LIN {X 0,Y 364.081,Z 519.091,A -85,B 0,C 180,E1 -13381.398,E2 -13381.398} C_VEL
LIN {X 0,Y 365.841,Z 526.741,A -85,B 0,C 180,E1 -13382.545,E2 -13382.545} C_VEL
LIN {X 0,Y 366.269,Z 538.243,A -85,B 0,C 180,E1 -13383.711,E2 -13383.711} C_VEL
LIN {X 0,Y 365.89,Z 556.59,A -85,B 0,C 180,E1 -13385.171,E2 -13385.171} C_VEL
LIN {X 0,Y 365.376,Z 561.748,A -85,B 0,C 180,E1 -13385.4,E2 -13385.4} C_VEL
LIN {X 0,Y 363.138,Z 602.546,A -85,B 0,C 180,E1 -13386.738,E2 -13386.738} C_VEL
LIN {X 0,Y 361.511,Z 662.702,A -85,B 0,C 180,E1 -13388.248,E2 -13388.248} C_VEL
LIN {X 0,Y 360.674,Z 677.145,A -85,B 0,C 180,E1 -13388.833,E2 -13388.833} C_VEL
LIN {X 0,Y 359.879,Z 691.511,A -85,B 0,C 180,E1 -13389.662,E2 -13389.662} C_VEL
LIN {X 0,Y 358.872,Z 705.143,A -85,B 0,C 180,E1 -13390.702,E2 -13390.702} C_VEL
LIN {X 0,Y 357.508,Z 721.974,A -85,B 0,C 180,E1 -13392.26,E2 -13392.26} C_VEL
LIN {X 0,Y 356.635,Z 733.015,A -85,B 0,C 180,E1 -13393.544,E2 -13393.544} C_VEL
LIN {X 0,Y 355.719,Z 743.896,A -85,B 0,C 180,E1 -13395.117,E2 -13395.117} C_VEL
LIN {X 0,Y 355.107,Z 752.022,A -85,B 0,C 180,E1 -13396.553,E2 -13396.553} C_VEL
LIN {X 0,Y 354.444,Z 759.998,A -85,B 0,C 180,E1 -13398.274,E2 -13398.274} C_VEL
LIN {X 0,Y 353.811,Z 767.392,A -85,B 0,C 180,E1 -13400.28,E2 -13400.28} C_VEL
LIN {X 0,Y 353.542,Z 772.311,A -85,B 0,C 180,E1 -13402.001,E2 -13402.001} C_VEL
LIN {X 0,Y 353.318,Z 776.57,A -85,B 0,C 180,E1 -13404.028,E2 -13404.028} C_VEL
LIN {X 0,Y 353.269,Z 778.692,A -85,B 0,C 180,E1 -13405.436,E2 -13405.436} C_VEL
LIN {X 0,Y 353.219,Z 780.707,A -85,B 0,C 180,E1 -13407.719,E2 -13407.719} C_VEL
LIN {X 0,Y 353.265,Z 781.559,A -85,B 0,C 180,E1 -13408.86,E2 -13408.86} C_VEL
LIN {X 0,Y 353.281,Z 782.044,A -85,B 0,C 180,E1 -13410,E2 -13410} C_VEL
LIN {X 0,Y 353.238,Z 782.141,A -85,B 0,C 180,E1 -13411.14,E2 -13411.14} C_VEL
LIN {X 0,Y 353.213,Z 781.212,A -85,B 0,C 180,E1 -13413.422,E2 -13413.422} C_VEL
LIN {X 0,Y 353.281,Z 778.816,A -85,B 0,C 180,E1 -13415.709,E2 -13415.709} C_VEL
LIN {X 0,Y 353.545,Z 774.903,A -85,B 0,C 180,E1 -13417.999,E2 -13417.999} C_VEL
LIN {X 0,Y 354.057,Z 769.384,A -85,B 0,C 180,E1 -13420.291,E2 -13420.291} C_VEL
LIN {X 0,Y 354.861,Z 763.039,A -85,B 0,C 180,E1 -13422.293,E2 -13422.293} C_VEL
LIN {X 0,Y 355.671,Z 756.174,A -85,B 0,C 180,E1 -13424.059,E2 -13424.059} C_VEL
LIN {X 0,Y 356.973,Z 746.863,A -85,B 0,C 180,E1 -13426,E2 -13426} C_VEL
LIN {X 0,Y 358.38,Z 736.943,A -85,B 0,C 180,E1 -13427.696,E2 -13427.696} C_VEL
LIN {X 0,Y 359.981,Z 725.962,A -85,B 0,C 180,E1 -13429.236,E2 -13429.236} C_VEL
LIN {X 0,Y 361.571,Z 714.167,A -85,B 0,C 180,E1 -13430.596,E2 -13430.596} C_VEL
LIN {X 0,Y 363.396,Z 700.647,A -85,B 0,C 180,E1 -13431.827,E2 -13431.827} C_VEL
LIN {X 0,Y 364.856,Z 687.097,A -85,B 0,C 180,E1 -13432.809,E2 -13432.809} C_VEL
LIN {X 0,Y 366.193,Z 673.662,A -85,B 0,C 180,E1 -13433.543,E2 -13433.543} C_VEL
LIN {X 0,Y 367.243,Z 659.343,A -85,B 0,C 180,E1 -13434.108,E2 -13434.108} C_VEL
LIN {X 0,Y 371.591,Z 579.823,A -85,B 0,C 180,E1 -13436.366,E2 -13436.366} C_VEL
LIN {X 0,Y 372.924,Z 556.68,A -85,B 0,C 180,E1 -13437.07,E2 -13437.07} C_VEL
LIN {X 0,Y 371.246,Z 544.885,A -85,B 0,C 180,E1 -13437.75,E2 -13437.75} C_VEL
LIN {X 0,Y 369.239,Z 535.063,A -85,B 0,C 180,E1 -13438.432,E2 -13438.432} C_VEL
LIN {X 0,Y 366.745,Z 529.791,A -85,B 0,C 180,E1 -13439.054,E2 -13439.054} C_VEL
LIN {X 0,Y 365.13,Z 522.109,A -85,B 0,C 180,E1 -13441.618,E2 -13441.618} C_VEL
LIN {X 0,Y 363.575,Z 515.996,A -85,B 0,C 180,E1 -13444.096,E2 -13444.096} C_VEL
LIN {X 0,Y 362.302,Z 511.752,A -85,B 0,C 180,E1 -13446.226,E2 -13446.226} C_VEL
LIN {X 0,Y 360.997,Z 507.772,A -85,B 0,C 180,E1 -13448.855,E2 -13448.855} C_VEL
LIN {X 0,Y 360.153,Z 504.97,A -85,B 0,C 180,E1 -13451.566,E2 -13451.566} C_VEL
LIN {X 0,Y 359.597,Z 503.898,A -85,B 0,C 180,E1 -13453.686,E2 -13453.686} C_VEL
LIN {X 0,Y 359.461,Z 503.658,A -85,B 0,C 180,E1 -13456.337,E2 -13456.337} C_VEL
LIN {X 0,Y 359.805,Z 504.291,A -85,B 0,C 180,E1 -13458.385,E2 -13458.385} C_VEL
LIN {X 0,Y 360.119,Z 505.331,A -85,B 0,C 180,E1 -13459.908,E2 -13459.908} C_VEL
LIN {X 0,Y 360.574,Z 506.767,A -85,B 0,C 180,E1 -13461.412,E2 -13461.412} C_VEL
LIN {X 0,Y 361.357,Z 509.306,A -85,B 0,C 180,E1 -13463.4,E2 -13463.4} C_VEL
LIN {X 0,Y 362.569,Z 513.268,A -85,B 0,C 180,E1 -13465.797,E2 -13465.797} C_VEL
LIN {X 0,Y 364.065,Z 519.255,A -85,B 0,C 180,E1 -13468.586,E2 -13468.586} C_VEL
LIN {X 0,Y 365.509,Z 526.31,A -85,B 0,C 180,E1 -13471.269,E2 -13471.269} C_VEL
LIN {X 0,Y 366.096,Z 531.225,A -85,B 0,C 180,E1 -13472.875,E2 -13472.875} C_VEL
LIN {X 0,Y 364.699,Z 538.089,A -85,B 0,C 180,E1 -13474.563,E2 -13474.563} C_VEL
LIN {X 0,Y 367.9,Z 551.216,A -85,B 0,C 180,E1 -13475.653,E2 -13475.653} C_VEL
LIN {X 0,Y 370.119,Z 562.832,A -85,B 0,C 180,E1 -13476.483,E2 -13476.483} C_VEL
LIN {X 0,Y 371.602,Z 573.765,A -85,B 0,C 180,E1 -13477.131,E2 -13477.131} C_VEL
LIN {X 0,Y 367.421,Z 636.034,A -85,B 0,C 180,E1 -13479.166,E2 -13479.166} C_VEL
LIN {X 0,Y 365.944,Z 658.464,A -85,B 0,C 180,E1 -13479.922,E2 -13479.922} C_VEL
LIN {X 0,Y 364.819,Z 671.855,A -85,B 0,C 180,E1 -13480.591,E2 -13480.591} C_VEL
LIN {X 0,Y 363.343,Z 686.293,A -85,B 0,C 180,E1 -13481.573,E2 -13481.573} C_VEL
LIN {X 0,Y 361.905,Z 698.511,A -85,B 0,C 180,E1 -13482.647,E2 -13482.647} C_VEL
LIN {X 0,Y 360.309,Z 710.785,A -85,B 0,C 180,E1 -13484.007,E2 -13484.007} C_VEL
LIN {X 0,Y 358.986,Z 719.938,A -85,B 0,C 180,E1 -13485.256,E2 -13485.256} C_VEL
LIN {X 0,Y 357.529,Z 729.94,A -85,B 0,C 180,E1 -13486.935,E2 -13486.935} C_VEL
LIN {X 0,Y 356.414,Z 738.093,A -85,B 0,C 180,E1 -13488.627,E2 -13488.627} C_VEL
LIN {X 0,Y 355.452,Z 744.674,A -85,B 0,C 180,E1 -13490.325,E2 -13490.325} C_VEL
LIN {X 0,Y 354.608,Z 750.579,A -85,B 0,C 180,E1 -13492.29,E2 -13492.29} C_VEL
LIN {X 0,Y 353.896,Z 755.09,A -85,B 0,C 180,E1 -13494.301,E2 -13494.301} C_VEL
LIN {X 0,Y 353.77,Z 756.988,A -85,B 0,C 180,E1 -13495.442,E2 -13495.442} C_VEL
LIN {X 0,Y 353.667,Z 758.395,A -85,B 0,C 180,E1 -13496.582,E2 -13496.582} C_VEL
LIN {X 0,Y 353.5,Z 759.383,A -85,B 0,C 180,E1 -13497.721,E2 -13497.721} C_VEL
LIN {X 0,Y 353.368,Z 759.956,A -85,B 0,C 180,E1 -13498.86,E2 -13498.86} C_VEL
LIN {X 0,Y 353.3,Z 760.1,A -85,B 0,C 180,E1 -13500,E2 -13500} C_VEL
LIN {X 0,Y 353.264,Z 759.775,A -85,B 0,C 180,E1 -13501.14,E2 -13501.14} C_VEL
LIN {X 0,Y 353.241,Z 759.032,A -85,B 0,C 180,E1 -13502.28,E2 -13502.28} C_VEL
LIN {X 0,Y 353.279,Z 757.868,A -85,B 0,C 180,E1 -13503.421,E2 -13503.421} C_VEL
LIN {X 0,Y 353.368,Z 755.247,A -85,B 0,C 180,E1 -13505.135,E2 -13505.135} C_VEL
LIN {X 0,Y 353.548,Z 751.024,A -85,B 0,C 180,E1 -13507.054,E2 -13507.054} C_VEL
LIN {X 0,Y 353.779,Z 746.7,A -85,B 0,C 180,E1 -13508.568,E2 -13508.568} C_VEL
LIN {X 0,Y 354.193,Z 740.537,A -85,B 0,C 180,E1 -13510.287,E2 -13510.287} C_VEL
LIN {X 0,Y 354.743,Z 732.82,A -85,B 0,C 180,E1 -13512.006,E2 -13512.006} C_VEL
LIN {X 0,Y 355.346,Z 724.997,A -85,B 0,C 180,E1 -13513.438,E2 -13513.438} C_VEL
LIN {X 0,Y 356.042,Z 715.561,A -85,B 0,C 180,E1 -13514.869,E2 -13514.869} C_VEL
LIN {X 0,Y 356.855,Z 705.267,A -85,B 0,C 180,E1 -13516.152,E2 -13516.152} C_VEL
LIN {X 0,Y 357.797,Z 694.015,A -85,B 0,C 180,E1 -13517.283,E2 -13517.283} C_VEL
LIN {X 0,Y 358.535,Z 681.676,A -85,B 0,C 180,E1 -13518.278,E2 -13518.278} C_VEL
LIN {X 0,Y 359.206,Z 669.161,A -85,B 0,C 180,E1 -13519.056,E2 -13519.056} C_VEL
LIN {X 0,Y 359.876,Z 654.808,A -85,B 0,C 180,E1 -13519.687,E2 -13519.687} C_VEL
LIN {X 0,Y 362.534,Z 570.248,A -85,B 0,C 180,E1 -13521.997,E2 -13521.997} C_VEL
LIN {X 0,Y 358.284,Z 539.518,A -85,B 0,C 180,E1 -13523.099,E2 -13523.099} C_VEL
LIN {X 0,Y 360.008,Z 522.356,A -85,B 0,C 180,E1 -13526.68,E2 -13526.68} C_VEL
LIN {X 0,Y 360.38,Z 516.609,A -85,B 0,C 180,E1 -13527.907,E2 -13527.907} C_VEL
LIN {X 0,Y 357.461,Z 503.16,A -85,B 0,C 180,E1 -13531.071,E2 -13531.071} C_VEL
LIN {X 0,Y 354.862,Z 491.409,A -85,B 0,C 180,E1 -13533.973,E2 -13533.973} C_VEL
LIN {X 0,Y 354.812,Z 491.413,A -85,B 0,C 180,E1 -13537.882,E2 -13537.882} C_VEL
LIN {X 0,Y 354.79,Z 491.414,A -85,B 0,C 180,E1 -13541.171,E2 -13541.171} C_VEL
LIN {X 0,Y 354.765,Z 491.415,A -85,B 0,C 180,E1 -13544.506,E2 -13544.506} C_VEL
LIN {X 0,Y 354.796,Z 491.417,A -85,B 0,C 180,E1 -13547.662,E2 -13547.662} C_VEL
LIN {X 0,Y 354.817,Z 491.409,A -85,B 0,C 180,E1 -13550.666,E2 -13550.666} C_VEL
LIN {X 0,Y 354.823,Z 491.408,A -85,B 0,C 180,E1 -13554.301,E2 -13554.301} C_VEL
LIN {X 0,Y 354.791,Z 491.417,A -85,B 0,C 180,E1 -13557.667,E2 -13557.667} C_VEL
LIN {X 0,Y 354.87,Z 491.402,A -85,B 0,C 180,E1 -13560.621,E2 -13560.621} C_VEL
LIN {X 0,Y 354.901,Z 491.399,A -85,B 0,C 180,E1 -13564.173,E2 -13564.173} C_VEL
LIN {X 0,Y 354.837,Z 491.409,A -85,B 0,C 180,E1 -13567.894,E2 -13567.894} C_VEL
LIN {X 0,Y 354.924,Z 491.398,A -85,B 0,C 180,E1 -13571.891,E2 -13571.891} C_VEL
LIN {X 0,Y 354.944,Z 491.395,A -85,B 0,C 180,E1 -13575.981,E2 -13575.981} C_VEL
LIN {X 0,Y 354.98,Z 491.392,A -85,B 0,C 180,E1 -13579.736,E2 -13579.736} C_VEL
LIN {X 0,Y 355.116,Z 491.373,A -85,B 0,C 180,E1 -13582.037,E2 -13582.037} C_VEL
LIN {X 0,Y 355.094,Z 491.374,A -85,B 0,C 180,E1 -13584.321,E2 -13584.321} C_VEL
LIN {X 0,Y 355.247,Z 491.359,A -85,B 0,C 180,E1 -13587.732,E2 -13587.732} C_VEL
LIN {X 0,Y 355.399,Z 491.338,A -85,B 0,C 180,E1 -13590,E2 -13590} C_VEL
LIN {X 0,Y 355.248,Z 491.355,A -85,B 0,C 180,E1 -13592.268,E2 -13592.268} C_VEL
LIN {X 0,Y 355.139,Z 491.37,A -85,B 0,C 180,E1 -13596.819,E2 -13596.819} C_VEL
LIN {X 0,Y 355.017,Z 491.387,A -85,B 0,C 180,E1 -13599.112,E2 -13599.112} C_VEL
LIN {X 0,Y 354.923,Z 491.396,A -85,B 0,C 180,E1 -13602.581,E2 -13602.581} C_VEL
LIN {X 0,Y 354.891,Z 491.4,A -85,B 0,C 180,E1 -13606.096,E2 -13606.096} C_VEL
LIN {X 0,Y 354.902,Z 491.398,A -85,B 0,C 180,E1 -13608.472,E2 -13608.472} C_VEL
LIN {X 0,Y 354.837,Z 491.407,A -85,B 0,C 180,E1 -13612.106,E2 -13612.106} C_VEL
LIN {X 0,Y 354.9,Z 491.4,A -85,B 0,C 180,E1 -13615.827,E2 -13615.827} C_VEL
LIN {X 0,Y 354.819,Z 491.412,A -85,B 0,C 180,E1 -13619.682,E2 -13619.682} C_VEL
LIN {X 0,Y 354.807,Z 491.413,A -85,B 0,C 180,E1 -13623.702,E2 -13623.702} C_VEL
LIN {X 0,Y 354.817,Z 491.411,A -85,B 0,C 180,E1 -13625.555,E2 -13625.555} C_VEL
LIN {X 0,Y 354.176,Z 491.492,A -85,B 0,C 180,E1 -13626.503,E2 -13626.503} C_VEL
LIN {X 0,Y 351.317,Z 491.849,A -85,B 0,C 180,E1 -13628.044,E2 -13628.044} C_VEL
LIN {X 0,Y 348.871,Z 492.156,A -85,B 0,C 180,E1 -13629.291,E2 -13629.291} C_VEL
LIN {X 0,Y 347.812,Z 492.282,A -85,B 0,C 180,E1 -13630.257,E2 -13630.257} C_VEL
LIN {X 0,Y 347.723,Z 492.291,A -85,B 0,C 180,E1 -13630.584,E2 -13630.584} C_VEL
LIN {X 0,Y 347.725,Z 492.298,A -85,B 0,C 180,E1 -13633.408,E2 -13633.408} C_VEL
LIN {X 0,Y 347.729,Z 492.293,A -85,B 0,C 180,E1 -13636.686,E2 -13636.686} C_VEL
LIN {X 0,Y 347.748,Z 492.289,A -85,B 0,C 180,E1 -13640.173,E2 -13640.173} C_VEL
LIN {X 0,Y 347.763,Z 492.289,A -85,B 0,C 180,E1 -13642.679,E2 -13642.679} C_VEL
LIN {X 0,Y 347.75,Z 492.293,A -85,B 0,C 180,E1 -13645.956,E2 -13645.956} C_VEL
LIN {X 0,Y 347.822,Z 492.393,A -85,B 0,C 180,E1 -13648.038,E2 -13648.038} C_VEL
LIN {X 0,Y 351.603,Z 508.967,A -85,B 0,C 180,E1 -13651.333,E2 -13651.333} C_VEL
LIN {X 0,Y 353.285,Z 517.769,A -85,B 0,C 180,E1 -13653.04,E2 -13653.04} C_VEL
LIN {X 0,Y 352.309,Z 533.649,A -85,B 0,C 180,E1 -13655.862,E2 -13655.862} C_VEL
LIN {X 0,Y 351.359,Z 548.377,A -85,B 0,C 180,E1 -13658.465,E2 -13658.465} C_VEL
LIN {X 0,Y 354.62,Z 574.143,A -85,B 0,C 180,E1 -13659.338,E2 -13659.338} C_VEL
LIN {X 0,Y 352.31,Z 659.734,A -85,B 0,C 180,E1 -13661.651,E2 -13661.651} C_VEL
LIN {X 0,Y 351.742,Z 672.287,A -85,B 0,C 180,E1 -13662.185,E2 -13662.185} C_VEL
LIN {X 0,Y 351.078,Z 685.288,A -85,B 0,C 180,E1 -13662.976,E2 -13662.976} C_VEL
LIN {X 0,Y 350.297,Z 697.868,A -85,B 0,C 180,E1 -13663.987,E2 -13663.987} C_VEL
LIN {X 0,Y 349.594,Z 709.123,A -85,B 0,C 180,E1 -13665.148,E2 -13665.148} C_VEL
LIN {X 0,Y 348.828,Z 719.418,A -85,B 0,C 180,E1 -13666.455,E2 -13666.455} C_VEL
LIN {X 0,Y 348.004,Z 729.556,A -85,B 0,C 180,E1 -13668.053,E2 -13668.053} C_VEL
LIN {X 0,Y 347.309,Z 738.483,A -85,B 0,C 180,E1 -13669.801,E2 -13669.801} C_VEL
LIN {X 0,Y 346.803,Z 745.567,A -85,B 0,C 180,E1 -13671.551,E2 -13671.551} C_VEL
LIN {X 0,Y 346.504,Z 752.191,A -85,B 0,C 180,E1 -13673.642,E2 -13673.642} C_VEL
LIN {X 0,Y 346.331,Z 756.244,A -85,B 0,C 180,E1 -13675.344,E2 -13675.344} C_VEL
LIN {X 0,Y 346.219,Z 758.381,A -85,B 0,C 180,E1 -13676.509,E2 -13676.509} C_VEL
LIN {X 0,Y 346.138,Z 760.082,A -85,B 0,C 180,E1 -13677.673,E2 -13677.673} C_VEL
LIN {X 0,Y 346.114,Z 761.316,A -85,B 0,C 180,E1 -13678.837,E2 -13678.837} C_VEL
LIN {X 0,Y 346.162,Z 762.087,A -85,B 0,C 180,E1 -13680,E2 -13680} C_VEL
LIN {X 0,Y 346.178,Z 762.447,A -85,B 0,C 180,E1 -13681.163,E2 -13681.163} C_VEL
LIN {X 0,Y 346.228,Z 762.363,A -85,B 0,C 180,E1 -13682.327,E2 -13682.327} C_VEL
LIN {X 0,Y 346.285,Z 761.812,A -85,B 0,C 180,E1 -13683.491,E2 -13683.491} C_VEL
LIN {X 0,Y 346.448,Z 760.844,A -85,B 0,C 180,E1 -13684.654,E2 -13684.654} C_VEL
LIN {X 0,Y 346.765,Z 759.439,A -85,B 0,C 180,E1 -13685.816,E2 -13685.816} C_VEL
LIN {X 0,Y 347.113,Z 756.474,A -85,B 0,C 180,E1 -13687.562,E2 -13687.562} C_VEL
LIN {X 0,Y 347.617,Z 752.407,A -85,B 0,C 180,E1 -13689.308,E2 -13689.308} C_VEL
LIN {X 0,Y 348.571,Z 746.1,A -85,B 0,C 180,E1 -13691.337,E2 -13691.337} C_VEL
LIN {X 0,Y 349.605,Z 739.197,A -85,B 0,C 180,E1 -13693.071,E2 -13693.071} C_VEL
LIN {X 0,Y 350.686,Z 732.203,A -85,B 0,C 180,E1 -13694.508,E2 -13694.508} C_VEL
LIN {X 0,Y 351.973,Z 723.754,A -85,B 0,C 180,E1 -13695.935,E2 -13695.935} C_VEL
LIN {X 0,Y 353.401,Z 713.472,A -85,B 0,C 180,E1 -13697.356,E2 -13697.356} C_VEL
LIN {X 0,Y 354.806,Z 701.968,A -85,B 0,C 180,E1 -13698.627,E2 -13698.627} C_VEL
LIN {X 0,Y 356.085,Z 690.911,A -85,B 0,C 180,E1 -13699.605,E2 -13699.605} C_VEL
LIN {X 0,Y 357.268,Z 678.942,A -85,B 0,C 180,E1 -13700.437,E2 -13700.437} C_VEL
LIN {X 0,Y 358.425,Z 664.617,A -85,B 0,C 180,E1 -13701.156,E2 -13701.156} C_VEL
LIN {X 0,Y 359.397,Z 645.914,A -85,B 0,C 180,E1 -13701.773,E2 -13701.773} C_VEL
LIN {X 0,Y 363.604,Z 576.847,A -85,B 0,C 180,E1 -13703.948,E2 -13703.948} C_VEL
LIN {X 0,Y 361.809,Z 565.369,A -85,B 0,C 180,E1 -13704.651,E2 -13704.651} C_VEL
LIN {X 0,Y 358.715,Z 551.015,A -85,B 0,C 180,E1 -13705.719,E2 -13705.719} C_VEL
LIN {X 0,Y 361.053,Z 533,A -85,B 0,C 180,E1 -13709.12,E2 -13709.12} C_VEL
LIN {X 0,Y 360.434,Z 527.37,A -85,B 0,C 180,E1 -13710.462,E2 -13710.462} C_VEL
LIN {X 0,Y 358.364,Z 518.355,A -85,B 0,C 180,E1 -13712.963,E2 -13712.963} C_VEL
LIN {X 0,Y 356.023,Z 510.706,A -85,B 0,C 180,E1 -13715.456,E2 -13715.456} C_VEL
LIN {X 0,Y 353.523,Z 504.31,A -85,B 0,C 180,E1 -13718.045,E2 -13718.045} C_VEL
LIN {X 0,Y 352.041,Z 500.989,A -85,B 0,C 180,E1 -13719.705,E2 -13719.705} C_VEL
LIN {X 0,Y 350.285,Z 497.307,A -85,B 0,C 180,E1 -13722.067,E2 -13722.067} C_VEL
LIN {X 0,Y 348.611,Z 494.858,A -85,B 0,C 180,E1 -13724.878,E2 -13724.878} C_VEL
LIN {X 0,Y 348.183,Z 493.986,A -85,B 0,C 180,E1 -13726.663,E2 -13726.663} C_VEL
LIN {X 0,Y 348.148,Z 493.877,A -85,B 0,C 180,E1 -13728.324,E2 -13728.324} C_VEL
LIN {X 0,Y 348.434,Z 494.54,A -85,B 0,C 180,E1 -13730.038,E2 -13730.038} C_VEL
LIN {X 0,Y 349.2,Z 495.784,A -85,B 0,C 180,E1 -13731.713,E2 -13731.713} C_VEL
LIN {X 0,Y 350.661,Z 497.181,A -85,B 0,C 180,E1 -13733.292,E2 -13733.292} C_VEL
LIN {X 0,Y 352.022,Z 500.297,A -85,B 0,C 180,E1 -13734.94,E2 -13734.94} C_VEL
LIN {X 0,Y 354.12,Z 503.338,A -85,B 0,C 180,E1 -13736.465,E2 -13736.465} C_VEL
LIN {X 0,Y 355.069,Z 505.854,A -85,B 0,C 180,E1 -13737.268,E2 -13737.268} C_VEL
LIN {X 0,Y 357.179,Z 515.611,A -85,B 0,C 180,E1 -13739.429,E2 -13739.429} C_VEL
LIN {X 0,Y 359.686,Z 525.404,A -85,B 0,C 180,E1 -13741.271,E2 -13741.271} C_VEL
LIN {X 0,Y 360.592,Z 529.454,A -85,B 0,C 180,E1 -13741.902,E2 -13741.902} C_VEL
LIN {X 0,Y 360.934,Z 538.418,A -85,B 0,C 180,E1 -13742.885,E2 -13742.885} C_VEL
LIN {X 0,Y 360.303,Z 557.83,A -85,B 0,C 180,E1 -13744.509,E2 -13744.509} C_VEL
LIN {X 0,Y 358.984,Z 575.75,A -85,B 0,C 180,E1 -13745.16,E2 -13745.16} C_VEL
LIN {X 0,Y 355.102,Z 645.539,A -85,B 0,C 180,E1 -13747.529,E2 -13747.529} C_VEL
LIN {X 0,Y 354.49,Z 664.577,A -85,B 0,C 180,E1 -13748.063,E2 -13748.063} C_VEL
LIN {X 0,Y 353.37,Z 685.73,A -85,B 0,C 180,E1 -13748.985,E2 -13748.985} C_VEL
LIN {X 0,Y 352.741,Z 699.341,A -85,B 0,C 180,E1 -13749.792,E2 -13749.792} C_VEL
LIN {X 0,Y 351.998,Z 711.641,A -85,B 0,C 180,E1 -13750.765,E2 -13750.765} C_VEL
LIN {X 0,Y 350.889,Z 723.393,A -85,B 0,C 180,E1 -13751.914,E2 -13751.914} C_VEL
LIN {X 0,Y 349.836,Z 735.116,A -85,B 0,C 180,E1 -13753.365,E2 -13753.365} C_VEL
LIN {X 0,Y 348.911,Z 744.702,A -85,B 0,C 180,E1 -13754.82,E2 -13754.82} C_VEL
LIN {X 0,Y 348.086,Z 753.98,A -85,B 0,C 180,E1 -13756.574,E2 -13756.574} C_VEL
LIN {X 0,Y 347.338,Z 761.578,A -85,B 0,C 180,E1 -13758.326,E2 -13758.326} C_VEL
LIN {X 0,Y 346.797,Z 767.665,A -85,B 0,C 180,E1 -13760.081,E2 -13760.081} C_VEL
LIN {X 0,Y 346.482,Z 772.437,A -85,B 0,C 180,E1 -13761.837,E2 -13761.837} C_VEL
LIN {X 0,Y 346.242,Z 776.829,A -85,B 0,C 180,E1 -13764.044,E2 -13764.044} C_VEL
LIN {X 0,Y 346.168,Z 778.641,A -85,B 0,C 180,E1 -13765.342,E2 -13765.342} C_VEL
LIN {X 0,Y 346.143,Z 779.77,A -85,B 0,C 180,E1 -13766.508,E2 -13766.508} C_VEL
LIN {X 0,Y 346.188,Z 781.742,A -85,B 0,C 180,E1 -13770,E2 -13770} C_VEL
LIN {X 0,Y 346.139,Z 781.899,A -85,B 0,C 180,E1 -13771.163,E2 -13771.163} C_VEL
LIN {X 0,Y 346.136,Z 781.068,A -85,B 0,C 180,E1 -13773.492,E2 -13773.492} C_VEL
LIN {X 0,Y 346.2,Z 778.748,A -85,B 0,C 180,E1 -13775.826,E2 -13775.826} C_VEL
LIN {X 0,Y 346.49,Z 774.922,A -85,B 0,C 180,E1 -13778.163,E2 -13778.163} C_VEL
LIN {X 0,Y 347.05,Z 769.498,A -85,B 0,C 180,E1 -13780.501,E2 -13780.501} C_VEL
LIN {X 0,Y 347.739,Z 764.234,A -85,B 0,C 180,E1 -13782.252,E2 -13782.252} C_VEL
LIN {X 0,Y 348.754,Z 756.717,A -85,B 0,C 180,E1 -13784.292,E2 -13784.292} C_VEL
LIN {X 0,Y 350.17,Z 747.367,A -85,B 0,C 180,E1 -13786.319,E2 -13786.319} C_VEL
LIN {X 0,Y 351.654,Z 737.617,A -85,B 0,C 180,E1 -13788.046,E2 -13788.046} C_VEL
LIN {X 0,Y 353.349,Z 726.834,A -85,B 0,C 180,E1 -13789.612,E2 -13789.612} C_VEL
LIN {X 0,Y 355.185,Z 714.25,A -85,B 0,C 180,E1 -13791.11,E2 -13791.11} C_VEL
LIN {X 0,Y 357.122,Z 700.915,A -85,B 0,C 180,E1 -13792.355,E2 -13792.355} C_VEL
LIN {X 0,Y 358.599,Z 688.224,A -85,B 0,C 180,E1 -13793.306,E2 -13793.306} C_VEL
LIN {X 0,Y 359.973,Z 675.311,A -85,B 0,C 180,E1 -13794.052,E2 -13794.052} C_VEL
LIN {X 0,Y 361.226,Z 660.185,A -85,B 0,C 180,E1 -13794.689,E2 -13794.689} C_VEL
LIN {X 0,Y 366.104,Z 578.96,A -85,B 0,C 180,E1 -13797.08,E2 -13797.08} C_VEL
LIN {X 0,Y 367.438,Z 558.125,A -85,B 0,C 180,E1 -13797.734,E2 -13797.734} C_VEL
LIN {X 0,Y 365.855,Z 546.557,A -85,B 0,C 180,E1 -13798.439,E2 -13798.439} C_VEL
LIN {X 0,Y 364.269,Z 538.562,A -85,B 0,C 180,E1 -13799.022,E2 -13799.022} C_VEL
LIN {X 0,Y 360.743,Z 531.845,A -85,B 0,C 180,E1 -13799.895,E2 -13799.895} C_VEL
LIN {X 0,Y 359.99,Z 530.14,A -85,B 0,C 180,E1 -13800.141,E2 -13800.141} C_VEL
LIN {X 0,Y 358.545,Z 523.573,A -85,B 0,C 180,E1 -13802.556,E2 -13802.556} C_VEL
LIN {X 0,Y 357.236,Z 518.532,A -85,B 0,C 180,E1 -13804.787,E2 -13804.787} C_VEL
LIN {X 0,Y 355.937,Z 514.083,A -85,B 0,C 180,E1 -13807.285,E2 -13807.285} C_VEL
LIN {X 0,Y 354.971,Z 511.227,A -85,B 0,C 180,E1 -13809.452,E2 -13809.452} C_VEL
LIN {X 0,Y 354.488,Z 509.58,A -85,B 0,C 180,E1 -13811.116,E2 -13811.116} C_VEL
LIN {X 0,Y 354.102,Z 508.504,A -85,B 0,C 180,E1 -13812.747,E2 -13812.747} C_VEL
LIN {X 0,Y 353.761,Z 507.836,A -85,B 0,C 180,E1 -13815.66,E2 -13815.66} C_VEL
LIN {X 0,Y 353.894,Z 508.145,A -85,B 0,C 180,E1 -13817.53,E2 -13817.53} C_VEL
LIN {X 0,Y 354.205,Z 508.884,A -85,B 0,C 180,E1 -13819.098,E2 -13819.098} C_VEL
LIN {X 0,Y 355.002,Z 511.73,A -85,B 0,C 180,E1 -13822.142,E2 -13822.142} C_VEL
LIN {X 0,Y 356.325,Z 515.972,A -85,B 0,C 180,E1 -13825.111,E2 -13825.111} C_VEL
LIN {X 0,Y 357.54,Z 521.052,A -85,B 0,C 180,E1 -13827.697,E2 -13827.697} C_VEL
LIN {X 0,Y 358.746,Z 526.559,A -85,B 0,C 180,E1 -13830.02,E2 -13830.02} C_VEL
LIN {X 0,Y 359.589,Z 532.152,A -85,B 0,C 180,E1 -13832.026,E2 -13832.026} C_VEL
LIN {X 0,Y 359.72,Z 534.169,A -85,B 0,C 180,E1 -13832.669,E2 -13832.669} C_VEL
LIN {X 0,Y 358.875,Z 537.88,A -85,B 0,C 180,E1 -13833.6,E2 -13833.6} C_VEL
LIN {X 0,Y 362.335,Z 552.245,A -85,B 0,C 180,E1 -13834.887,E2 -13834.887} C_VEL
LIN {X 0,Y 364.679,Z 564.501,A -85,B 0,C 180,E1 -13835.809,E2 -13835.809} C_VEL
LIN {X 0,Y 365.98,Z 575.262,A -85,B 0,C 180,E1 -13836.482,E2 -13836.482} C_VEL
LIN {X 0,Y 361.3,Z 639.592,A -85,B 0,C 180,E1 -13838.647,E2 -13838.647} C_VEL
LIN {X 0,Y 359.822,Z 659.996,A -85,B 0,C 180,E1 -13839.379,E2 -13839.379} C_VEL
LIN {X 0,Y 358.54,Z 674.125,A -85,B 0,C 180,E1 -13840.133,E2 -13840.133} C_VEL
LIN {X 0,Y 357.087,Z 687.256,A -85,B 0,C 180,E1 -13841.064,E2 -13841.064} C_VEL
LIN {X 0,Y 355.355,Z 700.576,A -85,B 0,C 180,E1 -13842.297,E2 -13842.297} C_VEL
LIN {X 0,Y 353.661,Z 712.54,A -85,B 0,C 180,E1 -13843.698,E2 -13843.698} C_VEL
LIN {X 0,Y 351.98,Z 723.242,A -85,B 0,C 180,E1 -13845.251,E2 -13845.251} C_VEL
LIN {X 0,Y 350.744,Z 731.23,A -85,B 0,C 180,E1 -13846.678,E2 -13846.678} C_VEL
LIN {X 0,Y 349.532,Z 739.131,A -85,B 0,C 180,E1 -13848.4,E2 -13848.4} C_VEL
LIN {X 0,Y 348.521,Z 745.536,A -85,B 0,C 180,E1 -13850.13,E2 -13850.13} C_VEL
LIN {X 0,Y 347.622,Z 751.391,A -85,B 0,C 180,E1 -13852.161,E2 -13852.161} C_VEL
LIN {X 0,Y 346.868,Z 755.699,A -85,B 0,C 180,E1 -13854.186,E2 -13854.186} C_VEL
LIN {X 0,Y 346.701,Z 757.483,A -85,B 0,C 180,E1 -13855.349,E2 -13855.349} C_VEL
LIN {X 0,Y 346.588,Z 758.824,A -85,B 0,C 180,E1 -13856.512,E2 -13856.512} C_VEL
LIN {X 0,Y 346.415,Z 759.761,A -85,B 0,C 180,E1 -13857.675,E2 -13857.675} C_VEL
LIN {X 0,Y 346.277,Z 760.278,A -85,B 0,C 180,E1 -13858.837,E2 -13858.837} C_VEL
LIN {X 0,Y 346.203,Z 760.322,A -85,B 0,C 180,E1 -13860,E2 -13860} C_VEL
LIN {X 0,Y 346.165,Z 759.937,A -85,B 0,C 180,E1 -13861.163,E2 -13861.163} C_VEL
LIN {X 0,Y 346.15,Z 759.134,A -85,B 0,C 180,E1 -13862.327,E2 -13862.327} C_VEL
LIN {X 0,Y 346.202,Z 757.898,A -85,B 0,C 180,E1 -13863.491,E2 -13863.491} C_VEL
LIN {X 0,Y 346.274,Z 755.174,A -85,B 0,C 180,E1 -13865.24,E2 -13865.24} C_VEL
LIN {X 0,Y 346.45,Z 751.134,A -85,B 0,C 180,E1 -13867.081,E2 -13867.081} C_VEL
LIN {X 0,Y 346.717,Z 746.383,A -85,B 0,C 180,E1 -13868.744,E2 -13868.744} C_VEL
LIN {X 0,Y 347.146,Z 740.044,A -85,B 0,C 180,E1 -13870.498,E2 -13870.498} C_VEL
LIN {X 0,Y 347.732,Z 732.156,A -85,B 0,C 180,E1 -13872.252,E2 -13872.252} C_VEL
LIN {X 0,Y 348.383,Z 724.152,A -85,B 0,C 180,E1 -13873.712,E2 -13873.712} C_VEL
LIN {X 0,Y 349.102,Z 714.497,A -85,B 0,C 180,E1 -13875.172,E2 -13875.172} C_VEL
LIN {X 0,Y 349.945,Z 703.85,A -85,B 0,C 180,E1 -13876.48,E2 -13876.48} C_VEL
LIN {X 0,Y 350.893,Z 692.254,A -85,B 0,C 180,E1 -13877.634,E2 -13877.634} C_VEL
LIN {X 0,Y 351.705,Z 679.403,A -85,B 0,C 180,E1 -13878.646,E2 -13878.646} C_VEL
LIN {X 0,Y 352.426,Z 666.025,A -85,B 0,C 180,E1 -13879.437,E2 -13879.437} C_VEL
LIN {X 0,Y 353.113,Z 652.429,A -85,B 0,C 180,E1 -13880.004,E2 -13880.004} C_VEL
LIN {X 0,Y 355.595,Z 570.586,A -85,B 0,C 180,E1 -13882.286,E2 -13882.286} C_VEL
LIN {X 0,Y 351.388,Z 539.457,A -85,B 0,C 180,E1 -13883.439,E2 -13883.439} C_VEL
LIN {X 0,Y 353.467,Z 520.198,A -85,B 0,C 180,E1 -13887.534,E2 -13887.534} C_VEL
LIN {X 0,Y 353.056,Z 515.786,A -85,B 0,C 180,E1 -13888.538,E2 -13888.538} C_VEL
LIN {X 0,Y 349.494,Z 499.955,A -85,B 0,C 180,E1 -13892.372,E2 -13892.372} C_VEL
LIN {X 0,Y 347.819,Z 492.285,A -85,B 0,C 180,E1 -13894.331,E2 -13894.331} C_VEL
LIN {X 0,Y 347.779,Z 492.288,A -85,B 0,C 180,E1 -13897.989,E2 -13897.989} C_VEL
LIN {X 0,Y 347.753,Z 492.293,A -85,B 0,C 180,E1 -13901.83,E2 -13901.83} C_VEL
LIN {X 0,Y 347.707,Z 492.296,A -85,B 0,C 180,E1 -13905.026,E2 -13905.026} C_VEL
LIN {X 0,Y 347.752,Z 492.289,A -85,B 0,C 180,E1 -13908.397,E2 -13908.397} C_VEL
LIN {X 0,Y 347.774,Z 492.288,A -85,B 0,C 180,E1 -13912.011,E2 -13912.011} C_VEL
LIN {X 0,Y 347.746,Z 492.296,A -85,B 0,C 180,E1 -13915.536,E2 -13915.536} C_VEL
LIN {X 0,Y 347.765,Z 492.292,A -85,B 0,C 180,E1 -13919.653,E2 -13919.653} C_VEL
LIN {X 0,Y 347.853,Z 492.277,A -85,B 0,C 180,E1 -13922.744,E2 -13922.744} C_VEL
LIN {X 0,Y 347.79,Z 492.285,A -85,B 0,C 180,E1 -13926.162,E2 -13926.162} C_VEL
LIN {X 0,Y 347.82,Z 492.283,A -85,B 0,C 180,E1 -13929.91,E2 -13929.91} C_VEL
LIN {X 0,Y 347.868,Z 492.275,A -85,B 0,C 180,E1 -13932.359,E2 -13932.359} C_VEL
LIN {X 0,Y 347.899,Z 492.272,A -85,B 0,C 180,E1 -13935.971,E2 -13935.971} C_VEL
LIN {X 0,Y 347.93,Z 492.273,A -85,B 0,C 180,E1 -13939.526,E2 -13939.526} C_VEL
LIN {X 0,Y 348.076,Z 492.251,A -85,B 0,C 180,E1 -13941.875,E2 -13941.875} C_VEL
LIN {X 0,Y 348.069,Z 492.25,A -85,B 0,C 180,E1 -13944.206,E2 -13944.206} C_VEL
LIN {X 0,Y 348.21,Z 492.236,A -85,B 0,C 180,E1 -13947.686,E2 -13947.686} C_VEL
LIN {X 0,Y 348.369,Z 492.213,A -85,B 0,C 180,E1 -13950,E2 -13950} C_VEL
LIN {X 0,Y 348.21,Z 492.232,A -85,B 0,C 180,E1 -13952.313,E2 -13952.313} C_VEL
LIN {X 0,Y 348.107,Z 492.247,A -85,B 0,C 180,E1 -13956.958,E2 -13956.958} C_VEL
LIN {X 0,Y 347.969,Z 492.267,A -85,B 0,C 180,E1 -13959.298,E2 -13959.298} C_VEL
LIN {X 0,Y 347.891,Z 492.273,A -85,B 0,C 180,E1 -13962.839,E2 -13962.839} C_VEL
LIN {X 0,Y 347.84,Z 492.278,A -85,B 0,C 180,E1 -13966.431,E2 -13966.431} C_VEL
LIN {X 0,Y 347.852,Z 492.278,A -85,B 0,C 180,E1 -13968.86,E2 -13968.86} C_VEL
LIN {X 0,Y 347.777,Z 492.286,A -85,B 0,C 180,E1 -13972.579,E2 -13972.579} C_VEL
LIN {X 0,Y 347.814,Z 492.285,A -85,B 0,C 180,E1 -13975.108,E2 -13975.108} C_VEL
LIN {X 0,Y 347.809,Z 492.285,A -85,B 0,C 180,E1 -13977.694,E2 -13977.694} C_VEL
LIN {X 0,Y 347.75,Z 492.289,A -85,B 0,C 180,E1 -13980.348,E2 -13980.348} C_VEL
LIN {X 0,Y 347.749,Z 492.29,A -85,B 0,C 180,E1 -13984.044,E2 -13984.044} C_VEL
LIN {X 0,Y 347.766,Z 492.294,A -85,B 0,C 180,E1 -13987.32,E2 -13987.32} C_VEL
LIN {X 0,Y 347.723,Z 492.291,A -85,B 0,C 180,E1 -13990.584,E2 -13990.584} C_VEL
LIN {X 0,Y 347.051,Z 492.38,A -85,B 0,C 180,E1 -13991.551,E2 -13991.551} C_VEL
LIN {X 0,Y 344.213,Z 492.735,A -85,B 0,C 180,E1 -13993.125,E2 -13993.125} C_VEL
LIN {X 0,Y 341.807,Z 493.037,A -85,B 0,C 180,E1 -13994.398,E2 -13994.398} C_VEL
LIN {X 0,Y 340.764,Z 493.165,A -85,B 0,C 180,E1 -13995.383,E2 -13995.383} C_VEL
LIN {X 0,Y 340.673,Z 493.173,A -85,B 0,C 180,E1 -13995.717,E2 -13995.717} C_VEL
LIN {X 0,Y 340.687,Z 493.17,A -85,B 0,C 180,E1 -13998.691,E2 -13998.691} C_VEL
LIN {X 0,Y 340.734,Z 493.165,A -85,B 0,C 180,E1 -14001.773,E2 -14001.773} C_VEL
LIN {X 0,Y 340.724,Z 493.169,A -85,B 0,C 180,E1 -14005.595,E2 -14005.595} C_VEL
LIN {X 0,Y 340.767,Z 493.302,A -85,B 0,C 180,E1 -14007.735,E2 -14007.735} C_VEL
LIN {X 0,Y 344.422,Z 509.197,A -85,B 0,C 180,E1 -14010.945,E2 -14010.945} C_VEL
LIN {X 0,Y 346.307,Z 518.612,A -85,B 0,C 180,E1 -14012.795,E2 -14012.795} C_VEL
LIN {X 0,Y 345.723,Z 529.343,A -85,B 0,C 180,E1 -14014.729,E2 -14014.729} C_VEL
LIN {X 0,Y 344.449,Z 548.373,A -85,B 0,C 180,E1 -14018.138,E2 -14018.138} C_VEL
LIN {X 0,Y 347.72,Z 574.625,A -85,B 0,C 180,E1 -14019.069,E2 -14019.069} C_VEL
LIN {X 0,Y 345.324,Z 660.254,A -85,B 0,C 180,E1 -14021.458,E2 -14021.458} C_VEL
LIN {X 0,Y 344.706,Z 673.242,A -85,B 0,C 180,E1 -14022.039,E2 -14022.039} C_VEL
LIN {X 0,Y 344.045,Z 686.015,A -85,B 0,C 180,E1 -14022.847,E2 -14022.847} C_VEL
LIN {X 0,Y 343.302,Z 697.649,A -85,B 0,C 180,E1 -14023.804,E2 -14023.804} C_VEL
LIN {X 0,Y 342.572,Z 708.733,A -85,B 0,C 180,E1 -14024.962,E2 -14024.962} C_VEL
LIN {X 0,Y 341.783,Z 719.298,A -85,B 0,C 180,E1 -14026.322,E2 -14026.322} C_VEL
LIN {X 0,Y 340.989,Z 728.669,A -85,B 0,C 180,E1 -14027.804,E2 -14027.804} C_VEL
LIN {X 0,Y 340.281,Z 737.792,A -85,B 0,C 180,E1 -14029.588,E2 -14029.588} C_VEL
LIN {X 0,Y 339.773,Z 745.101,A -85,B 0,C 180,E1 -14031.375,E2 -14031.375} C_VEL
LIN {X 0,Y 339.446,Z 751.191,A -85,B 0,C 180,E1 -14033.266,E2 -14033.266} C_VEL
LIN {X 0,Y 339.25,Z 756.081,A -85,B 0,C 180,E1 -14035.247,E2 -14035.247} C_VEL
LIN {X 0,Y 339.149,Z 758.305,A -85,B 0,C 180,E1 -14036.436,E2 -14036.436} C_VEL
LIN {X 0,Y 339.051,Z 760.063,A -85,B 0,C 180,E1 -14037.624,E2 -14037.624} C_VEL
LIN {X 0,Y 339.018,Z 761.39,A -85,B 0,C 180,E1 -14038.812,E2 -14038.812} C_VEL
LIN {X 0,Y 339.063,Z 762.225,A -85,B 0,C 180,E1 -14040,E2 -14040} C_VEL
LIN {X 0,Y 339.081,Z 762.634,A -85,B 0,C 180,E1 -14041.188,E2 -14041.188} C_VEL
LIN {X 0,Y 339.137,Z 762.628,A -85,B 0,C 180,E1 -14042.375,E2 -14042.375} C_VEL
LIN {X 0,Y 339.211,Z 762.152,A -85,B 0,C 180,E1 -14043.564,E2 -14043.564} C_VEL
LIN {X 0,Y 339.399,Z 761.241,A -85,B 0,C 180,E1 -14044.751,E2 -14044.751} C_VEL
LIN {X 0,Y 339.73,Z 759.908,A -85,B 0,C 180,E1 -14045.937,E2 -14045.937} C_VEL
LIN {X 0,Y 340.099,Z 757.044,A -85,B 0,C 180,E1 -14047.719,E2 -14047.719} C_VEL
LIN {X 0,Y 340.657,Z 753.088,A -85,B 0,C 180,E1 -14049.5,E2 -14049.5} C_VEL
LIN {X 0,Y 341.545,Z 747.934,A -85,B 0,C 180,E1 -14051.273,E2 -14051.273} C_VEL
LIN {X 0,Y 342.524,Z 741.456,A -85,B 0,C 180,E1 -14053.044,E2 -14053.044} C_VEL
LIN {X 0,Y 343.911,Z 733.382,A -85,B 0,C 180,E1 -14054.8,E2 -14054.8} C_VEL
LIN {X 0,Y 345.277,Z 725.132,A -85,B 0,C 180,E1 -14056.253,E2 -14056.253} C_VEL
LIN {X 0,Y 346.858,Z 714.617,A -85,B 0,C 180,E1 -14057.766,E2 -14057.766} C_VEL
LIN {X 0,Y 348.311,Z 704.157,A -85,B 0,C 180,E1 -14058.987,E2 -14058.987} C_VEL
LIN {X 0,Y 349.613,Z 693.548,A -85,B 0,C 180,E1 -14059.983,E2 -14059.983} C_VEL
LIN {X 0,Y 351.075,Z 680.042,A -85,B 0,C 180,E1 -14060.967,E2 -14060.967} C_VEL
LIN {X 0,Y 352.346,Z 665.458,A -85,B 0,C 180,E1 -14061.731,E2 -14061.731} C_VEL
LIN {X 0,Y 353.347,Z 648.75,A -85,B 0,C 180,E1 -14062.32,E2 -14062.32} C_VEL
LIN {X 0,Y 358.003,Z 578.864,A -85,B 0,C 180,E1 -14064.585,E2 -14064.585} C_VEL
LIN {X 0,Y 356.754,Z 569.615,A -85,B 0,C 180,E1 -14065.157,E2 -14065.157} C_VEL
LIN {X 0,Y 354.087,Z 556.328,A -85,B 0,C 180,E1 -14066.154,E2 -14066.154} C_VEL
LIN {X 0,Y 352.992,Z 551.281,A -85,B 0,C 180,E1 -14066.59,E2 -14066.59} C_VEL
LIN {X 0,Y 355.177,Z 535.491,A -85,B 0,C 180,E1 -14069.649,E2 -14069.649} C_VEL
LIN {X 0,Y 354.173,Z 528.615,A -85,B 0,C 180,E1 -14071.431,E2 -14071.431} C_VEL
LIN {X 0,Y 352.58,Z 521.373,A -85,B 0,C 180,E1 -14073.592,E2 -14073.592} C_VEL
LIN {X 0,Y 350.358,Z 514.195,A -85,B 0,C 180,E1 -14076.118,E2 -14076.118} C_VEL
LIN {X 0,Y 348.09,Z 508.242,A -85,B 0,C 180,E1 -14078.748,E2 -14078.748} C_VEL
LIN {X 0,Y 346.805,Z 505.336,A -85,B 0,C 180,E1 -14080.427,E2 -14080.427} C_VEL
LIN {X 0,Y 345.793,Z 502.82,A -85,B 0,C 180,E1 -14082.121,E2 -14082.121} C_VEL
LIN {X 0,Y 344.512,Z 500.855,A -85,B 0,C 180,E1 -14084.439,E2 -14084.439} C_VEL
LIN {X 0,Y 344.026,Z 499.715,A -85,B 0,C 180,E1 -14087.344,E2 -14087.344} C_VEL
LIN {X 0,Y 344.245,Z 500.055,A -85,B 0,C 180,E1 -14089.209,E2 -14089.209} C_VEL
LIN {X 0,Y 344.808,Z 501.025,A -85,B 0,C 180,E1 -14090.813,E2 -14090.813} C_VEL
LIN {X 0,Y 345.969,Z 502.404,A -85,B 0,C 180,E1 -14092.452,E2 -14092.452} C_VEL
LIN {X 0,Y 346.92,Z 503.636,A -85,B 0,C 180,E1 -14093.482,E2 -14093.482} C_VEL
LIN {X 0,Y 349.328,Z 507.782,A -85,B 0,C 180,E1 -14095.714,E2 -14095.714} C_VEL
LIN {X 0,Y 350.361,Z 509.645,A -85,B 0,C 180,E1 -14096.483,E2 -14096.483} C_VEL
LIN {X 0,Y 351.308,Z 514.331,A -85,B 0,C 180,E1 -14097.688,E2 -14097.688} C_VEL
LIN {X 0,Y 353.408,Z 523.826,A -85,B 0,C 180,E1 -14099.708,E2 -14099.708} C_VEL
LIN {X 0,Y 354.899,Z 530.089,A -85,B 0,C 180,E1 -14100.87,E2 -14100.87} C_VEL
LIN {X 0,Y 355.65,Z 534.066,A -85,B 0,C 180,E1 -14101.476,E2 -14101.476} C_VEL
LIN {X 0,Y 355.616,Z 542.496,A -85,B 0,C 180,E1 -14102.384,E2 -14102.384} C_VEL
LIN {X 0,Y 354.835,Z 558.727,A -85,B 0,C 180,E1 -14103.8,E2 -14103.8} C_VEL
LIN {X 0,Y 349.686,Z 639.02,A -85,B 0,C 180,E1 -14106.652,E2 -14106.652} C_VEL
LIN {X 0,Y 347.791,Z 675.973,A -85,B 0,C 180,E1 -14107.93,E2 -14107.93} C_VEL
LIN {X 0,Y 347.174,Z 689.109,A -85,B 0,C 180,E1 -14108.553,E2 -14108.553} C_VEL
LIN {X 0,Y 346.402,Z 701.618,A -85,B 0,C 180,E1 -14109.374,E2 -14109.374} C_VEL
LIN {X 0,Y 345.49,Z 713.638,A -85,B 0,C 180,E1 -14110.388,E2 -14110.388} C_VEL
LIN {X 0,Y 344.144,Z 726.143,A -85,B 0,C 180,E1 -14111.701,E2 -14111.701} C_VEL
LIN {X 0,Y 343.136,Z 736.254,A -85,B 0,C 180,E1 -14113.03,E2 -14113.03} C_VEL
LIN {X 0,Y 341.93,Z 747.282,A -85,B 0,C 180,E1 -14114.831,E2 -14114.831} C_VEL
LIN {X 0,Y 341.043,Z 755.971,A -85,B 0,C 180,E1 -14116.595,E2 -14116.595} C_VEL
LIN {X 0,Y 340.272,Z 763.066,A -85,B 0,C 180,E1 -14118.383,E2 -14118.383} C_VEL
LIN {X 0,Y 339.658,Z 769.639,A -85,B 0,C 180,E1 -14120.472,E2 -14120.472} C_VEL
LIN {X 0,Y 339.337,Z 773.919,A -85,B 0,C 180,E1 -14122.263,E2 -14122.263} C_VEL
LIN {X 0,Y 339.17,Z 777.084,A -85,B 0,C 180,E1 -14124.053,E2 -14124.053} C_VEL
LIN {X 0,Y 339.072,Z 778.592,A -85,B 0,C 180,E1 -14125.244,E2 -14125.244} C_VEL
LIN {X 0,Y 339.068,Z 779.676,A -85,B 0,C 180,E1 -14126.435,E2 -14126.435} C_VEL
LIN {X 0,Y 339.095,Z 781.427,A -85,B 0,C 180,E1 -14130,E2 -14130} C_VEL
LIN {X 0,Y 339.009,Z 781.46,A -85,B 0,C 180,E1 -14132.376,E2 -14132.376} C_VEL
LIN {X 0,Y 339.059,Z 780.921,A -85,B 0,C 180,E1 -14133.565,E2 -14133.565} C_VEL
LIN {X 0,Y 339.133,Z 778.696,A -85,B 0,C 180,E1 -14135.948,E2 -14135.948} C_VEL
LIN {X 0,Y 339.427,Z 774.965,A -85,B 0,C 180,E1 -14138.334,E2 -14138.334} C_VEL
LIN {X 0,Y 340.032,Z 769.637,A -85,B 0,C 180,E1 -14140.721,E2 -14140.721} C_VEL
LIN {X 0,Y 340.789,Z 764.484,A -85,B 0,C 180,E1 -14142.506,E2 -14142.506} C_VEL
LIN {X 0,Y 341.726,Z 758.238,A -85,B 0,C 180,E1 -14144.288,E2 -14144.288} C_VEL
LIN {X 0,Y 342.905,Z 750.742,A -85,B 0,C 180,E1 -14146.063,E2 -14146.063} C_VEL
LIN {X 0,Y 344.368,Z 741.749,A -85,B 0,C 180,E1 -14147.826,E2 -14147.826} C_VEL
LIN {X 0,Y 346.205,Z 730.893,A -85,B 0,C 180,E1 -14149.57,E2 -14149.57} C_VEL
LIN {X 0,Y 348,Z 720.016,A -85,B 0,C 180,E1 -14151.006,E2 -14151.006} C_VEL
LIN {X 0,Y 349.881,Z 708.066,A -85,B 0,C 180,E1 -14152.294,E2 -14152.294} C_VEL
LIN {X 0,Y 351.76,Z 694.449,A -85,B 0,C 180,E1 -14153.467,E2 -14153.467} C_VEL
LIN {X 0,Y 353.375,Z 680.92,A -85,B 0,C 180,E1 -14154.374,E2 -14154.374} C_VEL
LIN {X 0,Y 354.923,Z 665.774,A -85,B 0,C 180,E1 -14155.119,E2 -14155.119} C_VEL
LIN {X 0,Y 356.158,Z 646.071,A -85,B 0,C 180,E1 -14155.769,E2 -14155.769} C_VEL
LIN {X 0,Y 360.684,Z 579.154,A -85,B 0,C 180,E1 -14157.803,E2 -14157.803} C_VEL
LIN {X 0,Y 362.024,Z 559.019,A -85,B 0,C 180,E1 -14158.466,E2 -14158.466} C_VEL
LIN {X 0,Y 360.428,Z 547.203,A -85,B 0,C 180,E1 -14159.237,E2 -14159.237} C_VEL
LIN {X 0,Y 359.439,Z 542.409,A -85,B 0,C 180,E1 -14159.62,E2 -14159.62} C_VEL
LIN {X 0,Y 355.762,Z 535.133,A -85,B 0,C 180,E1 -14160.611,E2 -14160.611} C_VEL
LIN {X 0,Y 353.241,Z 530.558,A -85,B 0,C 180,E1 -14161.36,E2 -14161.36} C_VEL
LIN {X 0,Y 351.802,Z 524.164,A -85,B 0,C 180,E1 -14164.012,E2 -14164.012} C_VEL
LIN {X 0,Y 350.416,Z 519.225,A -85,B 0,C 180,E1 -14166.655,E2 -14166.655} C_VEL
LIN {X 0,Y 349.541,Z 516.486,A -85,B 0,C 180,E1 -14168.558,E2 -14168.558} C_VEL
LIN {X 0,Y 348.987,Z 514.71,A -85,B 0,C 180,E1 -14170.123,E2 -14170.123} C_VEL
LIN {X 0,Y 348.578,Z 513.316,A -85,B 0,C 180,E1 -14171.756,E2 -14171.756} C_VEL
LIN {X 0,Y 348.221,Z 512.461,A -85,B 0,C 180,E1 -14173.4,E2 -14173.4} C_VEL
LIN {X 0,Y 348.051,Z 512.101,A -85,B 0,C 180,E1 -14175.03,E2 -14175.03} C_VEL
LIN {X 0,Y 348.076,Z 512.173,A -85,B 0,C 180,E1 -14176.647,E2 -14176.647} C_VEL
LIN {X 0,Y 348.292,Z 512.691,A -85,B 0,C 180,E1 -14178.297,E2 -14178.297} C_VEL
LIN {X 0,Y 348.608,Z 513.77,A -85,B 0,C 180,E1 -14180.004,E2 -14180.004} C_VEL
LIN {X 0,Y 349.454,Z 516.755,A -85,B 0,C 180,E1 -14182.89,E2 -14182.89} C_VEL
LIN {X 0,Y 350.761,Z 521.31,A -85,B 0,C 180,E1 -14185.874,E2 -14185.874} C_VEL
LIN {X 0,Y 352.029,Z 527.19,A -85,B 0,C 180,E1 -14188.73,E2 -14188.73} C_VEL
LIN {X 0,Y 353.087,Z 533.267,A -85,B 0,C 180,E1 -14191.14,E2 -14191.14} C_VEL
LIN {X 0,Y 353.331,Z 537.139,A -85,B 0,C 180,E1 -14192.454,E2 -14192.454} C_VEL
LIN {X 0,Y 353.324,Z 537.933,A -85,B 0,C 180,E1 -14192.594,E2 -14192.594} C_VEL
LIN {X 0,Y 356.916,Z 553.056,A -85,B 0,C 180,E1 -14194.056,E2 -14194.056} C_VEL
LIN {X 0,Y 359.374,Z 566.605,A -85,B 0,C 180,E1 -14195.138,E2 -14195.138} C_VEL
LIN {X 0,Y 360.536,Z 577.027,A -85,B 0,C 180,E1 -14195.808,E2 -14195.808} C_VEL
LIN {X 0,Y 354.136,Z 658.212,A -85,B 0,C 180,E1 -14198.651,E2 -14198.651} C_VEL
LIN {X 0,Y 352.893,Z 671.376,A -85,B 0,C 180,E1 -14199.329,E2 -14199.329} C_VEL
LIN {X 0,Y 351.316,Z 684.601,A -85,B 0,C 180,E1 -14200.243,E2 -14200.243} C_VEL
LIN {X 0,Y 349.639,Z 697.567,A -85,B 0,C 180,E1 -14201.391,E2 -14201.391} C_VEL
LIN {X 0,Y 347.938,Z 708.974,A -85,B 0,C 180,E1 -14202.666,E2 -14202.666} C_VEL
LIN {X 0,Y 346.153,Z 719.408,A -85,B 0,C 180,E1 -14204.092,E2 -14204.092} C_VEL
LIN {X 0,Y 344.704,Z 728.032,A -85,B 0,C 180,E1 -14205.537,E2 -14205.537} C_VEL
LIN {X 0,Y 343.373,Z 736.573,A -85,B 0,C 180,E1 -14207.289,E2 -14207.289} C_VEL
LIN {X 0,Y 342.123,Z 743.508,A -85,B 0,C 180,E1 -14209.046,E2 -14209.046} C_VEL
LIN {X 0,Y 341.029,Z 749.89,A -85,B 0,C 180,E1 -14211.109,E2 -14211.109} C_VEL
LIN {X 0,Y 340.343,Z 754.091,A -85,B 0,C 180,E1 -14212.883,E2 -14212.883} C_VEL
LIN {X 0,Y 339.843,Z 756.3,A -85,B 0,C 180,E1 -14214.065,E2 -14214.065} C_VEL
LIN {X 0,Y 339.637,Z 758.003,A -85,B 0,C 180,E1 -14215.252,E2 -14215.252} C_VEL
LIN {X 0,Y 339.511,Z 759.283,A -85,B 0,C 180,E1 -14216.44,E2 -14216.44} C_VEL
LIN {X 0,Y 339.332,Z 760.153,A -85,B 0,C 180,E1 -14217.626,E2 -14217.626} C_VEL
LIN {X 0,Y 339.185,Z 760.565,A -85,B 0,C 180,E1 -14218.813,E2 -14218.813} C_VEL
LIN {X 0,Y 339.107,Z 760.538,A -85,B 0,C 180,E1 -14220,E2 -14220} C_VEL
LIN {X 0,Y 339.066,Z 760.094,A -85,B 0,C 180,E1 -14221.188,E2 -14221.188} C_VEL
LIN {X 0,Y 339.061,Z 759.229,A -85,B 0,C 180,E1 -14222.376,E2 -14222.376} C_VEL
LIN {X 0,Y 339.127,Z 757.885,A -85,B 0,C 180,E1 -14223.564,E2 -14223.564} C_VEL
LIN {X 0,Y 339.214,Z 754.468,A -85,B 0,C 180,E1 -14225.638,E2 -14225.638} C_VEL
LIN {X 0,Y 339.444,Z 749.528,A -85,B 0,C 180,E1 -14227.734,E2 -14227.734} C_VEL
LIN {X 0,Y 339.86,Z 742.88,A -85,B 0,C 180,E1 -14229.823,E2 -14229.823} C_VEL
LIN {X 0,Y 340.351,Z 735.639,A -85,B 0,C 180,E1 -14231.615,E2 -14231.615} C_VEL
LIN {X 0,Y 341.117,Z 726.669,A -85,B 0,C 180,E1 -14233.402,E2 -14233.402} C_VEL
LIN {X 0,Y 341.846,Z 716.785,A -85,B 0,C 180,E1 -14234.993,E2 -14234.993} C_VEL
LIN {X 0,Y 342.779,Z 706.281,A -85,B 0,C 180,E1 -14236.375,E2 -14236.375} C_VEL
LIN {X 0,Y 343.725,Z 695.252,A -85,B 0,C 180,E1 -14237.553,E2 -14237.553} C_VEL
LIN {X 0,Y 344.501,Z 683.176,A -85,B 0,C 180,E1 -14238.588,E2 -14238.588} C_VEL
LIN {X 0,Y 345.281,Z 669.844,A -85,B 0,C 180,E1 -14239.469,E2 -14239.469} C_VEL
LIN {X 0,Y 345.998,Z 655.86,A -85,B 0,C 180,E1 -14240.123,E2 -14240.123} C_VEL
LIN {X 0,Y 347.023,Z 624.112,A -85,B 0,C 180,E1 -14241.068,E2 -14241.068} C_VEL
LIN {X 0,Y 348.77,Z 571.488,A -85,B 0,C 180,E1 -14242.572,E2 -14242.572} C_VEL
LIN {X 0,Y 344.48,Z 539.395,A -85,B 0,C 180,E1 -14243.78,E2 -14243.78} C_VEL
LIN {X 0,Y 346.369,Z 522.413,A -85,B 0,C 180,E1 -14247.458,E2 -14247.458} C_VEL
LIN {X 0,Y 346.488,Z 519.374,A -85,B 0,C 180,E1 -14248.138,E2 -14248.138} C_VEL
LIN {X 0,Y 343.525,Z 505.783,A -85,B 0,C 180,E1 -14251.452,E2 -14251.452} C_VEL
LIN {X 0,Y 340.761,Z 493.163,A -85,B 0,C 180,E1 -14254.674,E2 -14254.674} C_VEL
LIN {X 0,Y 340.714,Z 493.166,A -85,B 0,C 180,E1 -14258.386,E2 -14258.386} C_VEL
LIN {X 0,Y 340.701,Z 493.169,A -85,B 0,C 180,E1 -14262.045,E2 -14262.045} C_VEL
LIN {X 0,Y 340.653,Z 493.174,A -85,B 0,C 180,E1 -14266.227,E2 -14266.227} C_VEL
LIN {X 0,Y 340.69,Z 493.173,A -85,B 0,C 180,E1 -14269.753,E2 -14269.753} C_VEL
LIN {X 0,Y 340.706,Z 493.17,A -85,B 0,C 180,E1 -14273.258,E2 -14273.258} C_VEL
LIN {X 0,Y 340.696,Z 493.169,A -85,B 0,C 180,E1 -14276.153,E2 -14276.153} C_VEL
LIN {X 0,Y 340.776,Z 493.158,A -85,B 0,C 180,E1 -14280.332,E2 -14280.332} C_VEL
LIN {X 0,Y 340.806,Z 493.156,A -85,B 0,C 180,E1 -14283.02,E2 -14283.02} C_VEL
LIN {X 0,Y 340.73,Z 493.165,A -85,B 0,C 180,E1 -14286.927,E2 -14286.927} C_VEL
LIN {X 0,Y 340.797,Z 493.156,A -85,B 0,C 180,E1 -14290.734,E2 -14290.734} C_VEL
LIN {X 0,Y 340.788,Z 493.16,A -85,B 0,C 180,E1 -14293.219,E2 -14293.219} C_VEL
LIN {X 0,Y 340.846,Z 493.15,A -85,B 0,C 180,E1 -14296.89,E2 -14296.89} C_VEL
LIN {X 0,Y 340.93,Z 493.139,A -85,B 0,C 180,E1 -14300.508,E2 -14300.508} C_VEL
LIN {X 0,Y 341.077,Z 493.122,A -85,B 0,C 180,E1 -14302.898,E2 -14302.898} C_VEL
LIN {X 0,Y 341.171,Z 493.113,A -85,B 0,C 180,E1 -14307.639,E2 -14307.639} C_VEL
LIN {X 0,Y 341.318,Z 493.092,A -85,B 0,C 180,E1 -14310,E2 -14310} C_VEL
LIN {X 0,Y 341.172,Z 493.109,A -85,B 0,C 180,E1 -14312.361,E2 -14312.361} C_VEL
LIN {X 0,Y 341.076,Z 493.123,A -85,B 0,C 180,E1 -14317.102,E2 -14317.102} C_VEL
LIN {X 0,Y 340.872,Z 493.146,A -85,B 0,C 180,E1 -14320.694,E2 -14320.694} C_VEL
LIN {X 0,Y 340.864,Z 493.147,A -85,B 0,C 180,E1 -14324.325,E2 -14324.325} C_VEL
LIN {X 0,Y 340.838,Z 493.15,A -85,B 0,C 180,E1 -14328.466,E2 -14328.466} C_VEL
LIN {X 0,Y 340.755,Z 493.162,A -85,B 0,C 180,E1 -14331.857,E2 -14331.857} C_VEL
LIN {X 0,Y 340.774,Z 493.161,A -85,B 0,C 180,E1 -14335.664,E2 -14335.664} C_VEL
LIN {X 0,Y 340.729,Z 493.164,A -85,B 0,C 180,E1 -14338.321,E2 -14338.321} C_VEL
LIN {X 0,Y 340.699,Z 493.171,A -85,B 0,C 180,E1 -14341.045,E2 -14341.045} C_VEL
LIN {X 0,Y 340.719,Z 493.171,A -85,B 0,C 180,E1 -14345.279,E2 -14345.279} C_VEL
LIN {X 0,Y 340.713,Z 493.166,A -85,B 0,C 180,E1 -14348.387,E2 -14348.387} C_VEL
LIN {X 0,Y 340.7,Z 493.168,A -85,B 0,C 180,E1 -14352.046,E2 -14352.046} C_VEL
LIN {X 0,Y 340.673,Z 493.173,A -85,B 0,C 180,E1 -14355.717,E2 -14355.717} C_VEL
LIN {X 0,Y 339.991,Z 493.258,A -85,B 0,C 180,E1 -14356.704,E2 -14356.704} C_VEL
LIN {X 0,Y 337.14,Z 493.611,A -85,B 0,C 180,E1 -14358.309,E2 -14358.309} C_VEL
LIN {X 0,Y 334.743,Z 493.913,A -85,B 0,C 180,E1 -14359.61,E2 -14359.61} C_VEL
LIN {X 0,Y 333.725,Z 494.037,A -85,B 0,C 180,E1 -14360.616,E2 -14360.616} C_VEL
LIN {X 0,Y 333.648,Z 494.049,A -85,B 0,C 180,E1 -14360.956,E2 -14360.956} C_VEL
LIN {X 0,Y 333.677,Z 494.043,A -85,B 0,C 180,E1 -14363.861,E2 -14363.861} C_VEL
LIN {X 0,Y 333.694,Z 494.06,A -85,B 0,C 180,E1 -14367.4,E2 -14367.4} C_VEL
LIN {X 0,Y 337.233,Z 509.461,A -85,B 0,C 180,E1 -14370.554,E2 -14370.554} C_VEL
LIN {X 0,Y 339.317,Z 519.534,A -85,B 0,C 180,E1 -14372.558,E2 -14372.558} C_VEL
LIN {X 0,Y 339.102,Z 526.638,A -85,B 0,C 180,E1 -14373.87,E2 -14373.87} C_VEL
LIN {X 0,Y 337.616,Z 547.609,A -85,B 0,C 180,E1 -14377.672,E2 -14377.672} C_VEL
LIN {X 0,Y 337.559,Z 549.011,A -85,B 0,C 180,E1 -14377.87,E2 -14377.87} C_VEL
LIN {X 0,Y 340.83,Z 575.589,A -85,B 0,C 180,E1 -14378.816,E2 -14378.816} C_VEL
LIN {X 0,Y 338.352,Z 660.158,A -85,B 0,C 180,E1 -14381.258,E2 -14381.258} C_VEL
LIN {X 0,Y 337.679,Z 673.857,A -85,B 0,C 180,E1 -14381.887,E2 -14381.887} C_VEL
LIN {X 0,Y 336.999,Z 686.518,A -85,B 0,C 180,E1 -14382.712,E2 -14382.712} C_VEL
LIN {X 0,Y 336.165,Z 698.827,A -85,B 0,C 180,E1 -14383.762,E2 -14383.762} C_VEL
LIN {X 0,Y 335.387,Z 710.672,A -85,B 0,C 180,E1 -14385.055,E2 -14385.055} C_VEL
LIN {X 0,Y 334.662,Z 720.192,A -85,B 0,C 180,E1 -14386.335,E2 -14386.335} C_VEL
LIN {X 0,Y 333.852,Z 729.422,A -85,B 0,C 180,E1 -14387.848,E2 -14387.848} C_VEL
LIN {X 0,Y 333.165,Z 738.481,A -85,B 0,C 180,E1 -14389.671,E2 -14389.671} C_VEL
LIN {X 0,Y 332.635,Z 745.679,A -85,B 0,C 180,E1 -14391.495,E2 -14391.495} C_VEL
LIN {X 0,Y 332.347,Z 751.594,A -85,B 0,C 180,E1 -14393.382,E2 -14393.382} C_VEL
LIN {X 0,Y 332.151,Z 755.887,A -85,B 0,C 180,E1 -14395.145,E2 -14395.145} C_VEL
LIN {X 0,Y 332.08,Z 758.221,A -85,B 0,C 180,E1 -14396.36,E2 -14396.36} C_VEL
LIN {X 0,Y 331.968,Z 760.03,A -85,B 0,C 180,E1 -14397.573,E2 -14397.573} C_VEL
LIN {X 0,Y 331.925,Z 761.412,A -85,B 0,C 180,E1 -14398.787,E2 -14398.787} C_VEL
LIN {X 0,Y 331.965,Z 762.352,A -85,B 0,C 180,E1 -14400,E2 -14400} C_VEL
LIN {X 0,Y 331.986,Z 762.819,A -85,B 0,C 180,E1 -14401.213,E2 -14401.213} C_VEL
LIN {X 0,Y 332.049,Z 762.87,A -85,B 0,C 180,E1 -14402.426,E2 -14402.426} C_VEL
LIN {X 0,Y 332.142,Z 762.497,A -85,B 0,C 180,E1 -14403.64,E2 -14403.64} C_VEL
LIN {X 0,Y 332.353,Z 761.642,A -85,B 0,C 180,E1 -14404.852,E2 -14404.852} C_VEL
LIN {X 0,Y 332.696,Z 760.358,A -85,B 0,C 180,E1 -14406.063,E2 -14406.063} C_VEL
LIN {X 0,Y 333.093,Z 757.612,A -85,B 0,C 180,E1 -14407.883,E2 -14407.883} C_VEL
LIN {X 0,Y 333.706,Z 753.805,A -85,B 0,C 180,E1 -14409.7,E2 -14409.7} C_VEL
LIN {X 0,Y 334.642,Z 748.808,A -85,B 0,C 180,E1 -14411.509,E2 -14411.509} C_VEL
LIN {X 0,Y 335.684,Z 742.481,A -85,B 0,C 180,E1 -14413.315,E2 -14413.315} C_VEL
LIN {X 0,Y 337.152,Z 734.595,A -85,B 0,C 180,E1 -14415.104,E2 -14415.104} C_VEL
LIN {X 0,Y 338.614,Z 726.615,A -85,B 0,C 180,E1 -14416.582,E2 -14416.582} C_VEL
LIN {X 0,Y 340.218,Z 716.943,A -85,B 0,C 180,E1 -14418.051,E2 -14418.051} C_VEL
LIN {X 0,Y 341.999,Z 704.918,A -85,B 0,C 180,E1 -14419.508,E2 -14419.508} C_VEL
LIN {X 0,Y 343.395,Z 694.595,A -85,B 0,C 180,E1 -14420.517,E2 -14420.517} C_VEL
LIN {X 0,Y 345.066,Z 680.45,A -85,B 0,C 180,E1 -14421.585,E2 -14421.585} C_VEL
LIN {X 0,Y 346.337,Z 666.858,A -85,B 0,C 180,E1 -14422.324,E2 -14422.324} C_VEL
LIN {X 0,Y 347.329,Z 651.787,A -85,B 0,C 180,E1 -14422.885,E2 -14422.885} C_VEL
LIN {X 0,Y 352.518,Z 579.664,A -85,B 0,C 180,E1 -14425.302,E2 -14425.302} C_VEL
LIN {X 0,Y 350.854,Z 568.306,A -85,B 0,C 180,E1 -14426.087,E2 -14426.087} C_VEL
LIN {X 0,Y 348.009,Z 554.517,A -85,B 0,C 180,E1 -14427.224,E2 -14427.224} C_VEL
LIN {X 0,Y 347.358,Z 551.744,A -85,B 0,C 180,E1 -14427.488,E2 -14427.488} C_VEL
LIN {X 0,Y 349.326,Z 539.626,A -85,B 0,C 180,E1 -14429.867,E2 -14429.867} C_VEL
LIN {X 0,Y 348.97,Z 534.798,A -85,B 0,C 180,E1 -14431.085,E2 -14431.085} C_VEL
LIN {X 0,Y 347.393,Z 526.722,A -85,B 0,C 180,E1 -14433.481,E2 -14433.481} C_VEL
LIN {X 0,Y 345.824,Z 520.703,A -85,B 0,C 180,E1 -14435.619,E2 -14435.619} C_VEL
LIN {X 0,Y 343.716,Z 514.473,A -85,B 0,C 180,E1 -14438.325,E2 -14438.325} C_VEL
LIN {X 0,Y 342.17,Z 510.671,A -85,B 0,C 180,E1 -14440.539,E2 -14440.539} C_VEL
LIN {X 0,Y 340.998,Z 507.678,A -85,B 0,C 180,E1 -14442.854,E2 -14442.854} C_VEL
LIN {X 0,Y 340.079,Z 506.103,A -85,B 0,C 180,E1 -14445.361,E2 -14445.361} C_VEL
LIN {X 0,Y 339.956,Z 505.603,A -85,B 0,C 180,E1 -14446.983,E2 -14446.983} C_VEL
LIN {X 0,Y 340.152,Z 505.776,A -85,B 0,C 180,E1 -14448.611,E2 -14448.611} C_VEL
LIN {X 0,Y 340.659,Z 506.562,A -85,B 0,C 180,E1 -14450.242,E2 -14450.242} C_VEL
LIN {X 0,Y 341.729,Z 507.894,A -85,B 0,C 180,E1 -14451.904,E2 -14451.904} C_VEL
LIN {X 0,Y 343.136,Z 509.905,A -85,B 0,C 180,E1 -14453.561,E2 -14453.561} C_VEL
LIN {X 0,Y 345.508,Z 513.908,A -85,B 0,C 180,E1 -14455.687,E2 -14455.687} C_VEL
LIN {X 0,Y 346.33,Z 515.511,A -85,B 0,C 180,E1 -14456.305,E2 -14456.305} C_VEL
LIN {X 0,Y 347.361,Z 521.88,A -85,B 0,C 180,E1 -14457.873,E2 -14457.873} C_VEL
LIN {X 0,Y 349.704,Z 532.418,A -85,B 0,C 180,E1 -14460.057,E2 -14460.057} C_VEL
LIN {X 0,Y 350.563,Z 537.501,A -85,B 0,C 180,E1 -14460.882,E2 -14460.882} C_VEL
LIN {X 0,Y 350.41,Z 544.924,A -85,B 0,C 180,E1 -14461.705,E2 -14461.705} C_VEL
LIN {X 0,Y 349.585,Z 558.26,A -85,B 0,C 180,E1 -14462.923,E2 -14462.923} C_VEL
LIN {X 0,Y 349.459,Z 562.438,A -85,B 0,C 180,E1 -14463.137,E2 -14463.137} C_VEL
LIN {X 0,Y 343.305,Z 649.657,A -85,B 0,C 180,E1 -14466.312,E2 -14466.312} C_VEL
LIN {X 0,Y 341.674,Z 680.106,A -85,B 0,C 180,E1 -14467.434,E2 -14467.434} C_VEL
LIN {X 0,Y 340.933,Z 692.654,A -85,B 0,C 180,E1 -14468.123,E2 -14468.123} C_VEL
LIN {X 0,Y 339.845,Z 706.292,A -85,B 0,C 180,E1 -14469.126,E2 -14469.126} C_VEL
LIN {X 0,Y 338.645,Z 718.659,A -85,B 0,C 180,E1 -14470.291,E2 -14470.291} C_VEL
LIN {X 0,Y 337.313,Z 729.968,A -85,B 0,C 180,E1 -14471.631,E2 -14471.631} C_VEL
LIN {X 0,Y 336.252,Z 739.342,A -85,B 0,C 180,E1 -14472.985,E2 -14472.985} C_VEL
LIN {X 0,Y 335.137,Z 748.215,A -85,B 0,C 180,E1 -14474.524,E2 -14474.524} C_VEL
LIN {X 0,Y 334.154,Z 756.558,A -85,B 0,C 180,E1 -14476.313,E2 -14476.313} C_VEL
LIN {X 0,Y 333.324,Z 763.522,A -85,B 0,C 180,E1 -14478.137,E2 -14478.137} C_VEL
LIN {X 0,Y 332.633,Z 769.9,A -85,B 0,C 180,E1 -14480.269,E2 -14480.269} C_VEL
LIN {X 0,Y 332.282,Z 774.039,A -85,B 0,C 180,E1 -14482.098,E2 -14482.098} C_VEL
LIN {X 0,Y 332.086,Z 777.31,A -85,B 0,C 180,E1 -14484.083,E2 -14484.083} C_VEL
LIN {X 0,Y 331.971,Z 779.596,A -85,B 0,C 180,E1 -14486.359,E2 -14486.359} C_VEL
LIN {X 0,Y 332.002,Z 781.104,A -85,B 0,C 180,E1 -14490,E2 -14490} C_VEL
LIN {X 0,Y 331.925,Z 781.235,A -85,B 0,C 180,E1 -14492.427,E2 -14492.427} C_VEL
LIN {X 0,Y 331.962,Z 780.747,A -85,B 0,C 180,E1 -14493.642,E2 -14493.642} C_VEL
LIN {X 0,Y 332.043,Z 778.657,A -85,B 0,C 180,E1 -14496.075,E2 -14496.075} C_VEL
LIN {X 0,Y 332.381,Z 775.03,A -85,B 0,C 180,E1 -14498.512,E2 -14498.512} C_VEL
LIN {X 0,Y 333.033,Z 769.81,A -85,B 0,C 180,E1 -14500.949,E2 -14500.949} C_VEL
LIN {X 0,Y 333.849,Z 764.778,A -85,B 0,C 180,E1 -14502.77,E2 -14502.77} C_VEL
LIN {X 0,Y 334.988,Z 757.129,A -85,B 0,C 180,E1 -14504.998,E2 -14504.998} C_VEL
LIN {X 0,Y 336.606,Z 748.545,A -85,B 0,C 180,E1 -14506.996,E2 -14506.996} C_VEL
LIN {X 0,Y 338.262,Z 739.219,A -85,B 0,C 180,E1 -14508.787,E2 -14508.787} C_VEL
LIN {X 0,Y 340.182,Z 728.924,A -85,B 0,C 180,E1 -14510.404,E2 -14510.404} C_VEL
LIN {X 0,Y 342.046,Z 717.856,A -85,B 0,C 180,E1 -14511.847,E2 -14511.847} C_VEL
LIN {X 0,Y 344.367,Z 704.099,A -85,B 0,C 180,E1 -14513.277,E2 -14513.277} C_VEL
LIN {X 0,Y 346.083,Z 692.07,A -85,B 0,C 180,E1 -14514.282,E2 -14514.282} C_VEL
LIN {X 0,Y 347.69,Z 679.412,A -85,B 0,C 180,E1 -14515.118,E2 -14515.118} C_VEL
LIN {X 0,Y 349.222,Z 664.662,A -85,B 0,C 180,E1 -14515.838,E2 -14515.838} C_VEL
LIN {X 0,Y 350.933,Z 639.592,A -85,B 0,C 180,E1 -14516.662,E2 -14516.662} C_VEL
LIN {X 0,Y 356.076,Z 571.195,A -85,B 0,C 180,E1 -14518.831,E2 -14518.831} C_VEL
LIN {X 0,Y 356.822,Z 560.613,A -85,B 0,C 180,E1 -14519.197,E2 -14519.197} C_VEL
LIN {X 0,Y 355.243,Z 548.301,A -85,B 0,C 180,E1 -14520.046,E2 -14520.046} C_VEL
LIN {X 0,Y 354.691,Z 546.146,A -85,B 0,C 180,E1 -14520.252,E2 -14520.252} C_VEL
LIN {X 0,Y 351.301,Z 539.473,A -85,B 0,C 180,E1 -14521.226,E2 -14521.226} C_VEL
LIN {X 0,Y 348.696,Z 535.001,A -85,B 0,C 180,E1 -14522.003,E2 -14522.003} C_VEL
LIN {X 0,Y 346.501,Z 531.004,A -85,B 0,C 180,E1 -14522.764,E2 -14522.764} C_VEL
LIN {X 0,Y 345.173,Z 525.337,A -85,B 0,C 180,E1 -14525.469,E2 -14525.469} C_VEL
LIN {X 0,Y 344.093,Z 521.681,A -85,B 0,C 180,E1 -14527.788,E2 -14527.788} C_VEL
LIN {X 0,Y 343.083,Z 518.391,A -85,B 0,C 180,E1 -14530.717,E2 -14530.717} C_VEL
LIN {X 0,Y 342.665,Z 517.093,A -85,B 0,C 180,E1 -14532.596,E2 -14532.596} C_VEL
LIN {X 0,Y 342.401,Z 516.49,A -85,B 0,C 180,E1 -14534.257,E2 -14534.257} C_VEL
LIN {X 0,Y 342.407,Z 516.584,A -85,B 0,C 180,E1 -14537.364,E2 -14537.364} C_VEL
LIN {X 0,Y 342.706,Z 517.481,A -85,B 0,C 180,E1 -14539.357,E2 -14539.357} C_VEL
LIN {X 0,Y 343.362,Z 519.956,A -85,B 0,C 180,E1 -14542.117,E2 -14542.117} C_VEL
LIN {X 0,Y 344.362,Z 523.4,A -85,B 0,C 180,E1 -14544.722,E2 -14544.722} C_VEL
LIN {X 0,Y 345.301,Z 527.565,A -85,B 0,C 180,E1 -14547.088,E2 -14547.088} C_VEL
LIN {X 0,Y 346.311,Z 532.86,A -85,B 0,C 180,E1 -14549.513,E2 -14549.513} C_VEL
LIN {X 0,Y 347.074,Z 537.564,A -85,B 0,C 180,E1 -14551.287,E2 -14551.287} C_VEL
LIN {X 0,Y 348.996,Z 542.331,A -85,B 0,C 180,E1 -14551.99,E2 -14551.99} C_VEL
LIN {X 0,Y 352.126,Z 556.395,A -85,B 0,C 180,E1 -14553.401,E2 -14553.401} C_VEL
LIN {X 0,Y 354.183,Z 568.601,A -85,B 0,C 180,E1 -14554.416,E2 -14554.416} C_VEL
LIN {X 0,Y 355.21,Z 578.385,A -85,B 0,C 180,E1 -14555.08,E2 -14555.08} C_VEL
LIN {X 0,Y 349.747,Z 642.203,A -85,B 0,C 180,E1 -14557.36,E2 -14557.36} C_VEL
LIN {X 0,Y 348.178,Z 660.549,A -85,B 0,C 180,E1 -14558.073,E2 -14558.073} C_VEL
LIN {X 0,Y 346.596,Z 675.216,A -85,B 0,C 180,E1 -14558.904,E2 -14558.904} C_VEL
LIN {X 0,Y 344.934,Z 688.171,A -85,B 0,C 180,E1 -14559.874,E2 -14559.874} C_VEL
LIN {X 0,Y 342.934,Z 701.516,A -85,B 0,C 180,E1 -14561.169,E2 -14561.169} C_VEL
LIN {X 0,Y 340.989,Z 713.25,A -85,B 0,C 180,E1 -14562.611,E2 -14562.611} C_VEL
LIN {X 0,Y 339.18,Z 722.976,A -85,B 0,C 180,E1 -14564.065,E2 -14564.065} C_VEL
LIN {X 0,Y 337.458,Z 732.523,A -85,B 0,C 180,E1 -14565.835,E2 -14565.835} C_VEL
LIN {X 0,Y 336.11,Z 740.189,A -85,B 0,C 180,E1 -14567.624,E2 -14567.624} C_VEL
LIN {X 0,Y 334.969,Z 745.575,A -85,B 0,C 180,E1 -14569.115,E2 -14569.115} C_VEL
LIN {X 0,Y 334.086,Z 750.765,A -85,B 0,C 180,E1 -14570.922,E2 -14570.922} C_VEL
LIN {X 0,Y 333.335,Z 754.806,A -85,B 0,C 180,E1 -14572.732,E2 -14572.732} C_VEL
LIN {X 0,Y 332.821,Z 756.887,A -85,B 0,C 180,E1 -14573.939,E2 -14573.939} C_VEL
LIN {X 0,Y 332.575,Z 758.526,A -85,B 0,C 180,E1 -14575.151,E2 -14575.151} C_VEL
LIN {X 0,Y 332.434,Z 759.748,A -85,B 0,C 180,E1 -14576.364,E2 -14576.364} C_VEL
LIN {X 0,Y 332.247,Z 760.519,A -85,B 0,C 180,E1 -14577.575,E2 -14577.575} C_VEL
LIN {X 0,Y 332.093,Z 760.845,A -85,B 0,C 180,E1 -14578.787,E2 -14578.787} C_VEL
LIN {X 0,Y 332.01,Z 760.754,A -85,B 0,C 180,E1 -14580,E2 -14580} C_VEL
LIN {X 0,Y 331.97,Z 760.244,A -85,B 0,C 180,E1 -14581.213,E2 -14581.213} C_VEL
LIN {X 0,Y 331.976,Z 759.275,A -85,B 0,C 180,E1 -14582.427,E2 -14582.427} C_VEL
LIN {X 0,Y 332.053,Z 757.857,A -85,B 0,C 180,E1 -14583.64,E2 -14583.64} C_VEL
LIN {X 0,Y 332.107,Z 754.7,A -85,B 0,C 180,E1 -14585.56,E2 -14585.56} C_VEL
LIN {X 0,Y 332.291,Z 750.803,A -85,B 0,C 180,E1 -14587.291,E2 -14587.291} C_VEL
LIN {X 0,Y 332.643,Z 744.509,A -85,B 0,C 180,E1 -14589.424,E2 -14589.424} C_VEL
LIN {X 0,Y 333.138,Z 737.583,A -85,B 0,C 180,E1 -14591.253,E2 -14591.253} C_VEL
LIN {X 0,Y 333.927,Z 728.985,A -85,B 0,C 180,E1 -14593.076,E2 -14593.076} C_VEL
LIN {X 0,Y 334.508,Z 719.46,A -85,B 0,C 180,E1 -14594.727,E2 -14594.727} C_VEL
LIN {X 0,Y 335.592,Z 708.405,A -85,B 0,C 180,E1 -14596.266,E2 -14596.266} C_VEL
LIN {X 0,Y 336.617,Z 696.349,A -85,B 0,C 180,E1 -14597.622,E2 -14597.622} C_VEL
LIN {X 0,Y 337.406,Z 684.524,A -85,B 0,C 180,E1 -14598.678,E2 -14598.678} C_VEL
LIN {X 0,Y 338.27,Z 670.379,A -85,B 0,C 180,E1 -14599.653,E2 -14599.653} C_VEL
LIN {X 0,Y 339.039,Z 655.832,A -85,B 0,C 180,E1 -14600.357,E2 -14600.357} C_VEL
LIN {X 0,Y 340.121,Z 623.8,A -85,B 0,C 180,E1 -14601.344,E2 -14601.344} C_VEL
LIN {X 0,Y 341.919,Z 572.039,A -85,B 0,C 180,E1 -14602.882,E2 -14602.882} C_VEL
LIN {X 0,Y 337.628,Z 539.287,A -85,B 0,C 180,E1 -14604.142,E2 -14604.142} C_VEL
LIN {X 0,Y 339.508,Z 522.885,A -85,B 0,C 180,E1 -14607.76,E2 -14607.76} C_VEL
LIN {X 0,Y 339.446,Z 519.954,A -85,B 0,C 180,E1 -14608.437,E2 -14608.437} C_VEL
LIN {X 0,Y 336.061,Z 504.794,A -85,B 0,C 180,E1 -14612.227,E2 -14612.227} C_VEL
LIN {X 0,Y 333.707,Z 494.042,A -85,B 0,C 180,E1 -14615.04,E2 -14615.04} C_VEL
LIN {X 0,Y 333.656,Z 494.045,A -85,B 0,C 180,E1 -14618.798,E2 -14618.798} C_VEL
LIN {X 0,Y 333.634,Z 494.048,A -85,B 0,C 180,E1 -14622.5,E2 -14622.5} C_VEL
LIN {X 0,Y 333.598,Z 494.055,A -85,B 0,C 180,E1 -14625.955,E2 -14625.955} C_VEL
LIN {X 0,Y 333.649,Z 494.049,A -85,B 0,C 180,E1 -14629.315,E2 -14629.315} C_VEL
LIN {X 0,Y 333.666,Z 494.046,A -85,B 0,C 180,E1 -14633.168,E2 -14633.168} C_VEL
LIN {X 0,Y 333.64,Z 494.047,A -85,B 0,C 180,E1 -14636.792,E2 -14636.792} C_VEL
LIN {X 0,Y 333.704,Z 494.043,A -85,B 0,C 180,E1 -14639.71,E2 -14639.71} C_VEL
LIN {X 0,Y 333.745,Z 494.034,A -85,B 0,C 180,E1 -14642.401,E2 -14642.401} C_VEL
LIN {X 0,Y 333.728,Z 494.038,A -85,B 0,C 180,E1 -14645.091,E2 -14645.091} C_VEL
LIN {X 0,Y 333.689,Z 494.042,A -85,B 0,C 180,E1 -14649.02,E2 -14649.02} C_VEL
LIN {X 0,Y 333.796,Z 494.033,A -85,B 0,C 180,E1 -14651.589,E2 -14651.589} C_VEL
LIN {X 0,Y 333.81,Z 494.031,A -85,B 0,C 180,E1 -14655.576,E2 -14655.576} C_VEL
LIN {X 0,Y 333.835,Z 494.025,A -85,B 0,C 180,E1 -14659.078,E2 -14659.078} C_VEL
LIN {X 0,Y 334.027,Z 493.999,A -85,B 0,C 180,E1 -14662.747,E2 -14662.747} C_VEL
LIN {X 0,Y 333.813,Z 494.029,A -85,B 0,C 180,E1 -14665.169,E2 -14665.169} C_VEL
LIN {X 0,Y 334.133,Z 493.99,A -85,B 0,C 180,E1 -14667.589,E2 -14667.589} C_VEL
LIN {X 0,Y 334.268,Z 493.97,A -85,B 0,C 180,E1 -14670,E2 -14670} C_VEL
LIN {X 0,Y 334.109,Z 493.988,A -85,B 0,C 180,E1 -14672.411,E2 -14672.411} C_VEL
LIN {X 0,Y 334.026,Z 494.003,A -85,B 0,C 180,E1 -14677.252,E2 -14677.252} C_VEL
LIN {X 0,Y 333.835,Z 494.024,A -85,B 0,C 180,E1 -14680.922,E2 -14680.922} C_VEL
LIN {X 0,Y 333.809,Z 494.026,A -85,B 0,C 180,E1 -14684.634,E2 -14684.634} C_VEL
LIN {X 0,Y 333.797,Z 494.028,A -85,B 0,C 180,E1 -14688.655,E2 -14688.655} C_VEL
LIN {X 0,Y 333.694,Z 494.04,A -85,B 0,C 180,E1 -14692.278,E2 -14692.278} C_VEL
LIN {X 0,Y 333.736,Z 494.035,A -85,B 0,C 180,E1 -14696.246,E2 -14696.246} C_VEL
LIN {X 0,Y 333.691,Z 494.043,A -85,B 0,C 180,E1 -14698.974,E2 -14698.974} C_VEL
LIN {X 0,Y 333.644,Z 494.047,A -85,B 0,C 180,E1 -14702.587,E2 -14702.587} C_VEL
LIN {X 0,Y 333.678,Z 494.042,A -85,B 0,C 180,E1 -14706.139,E2 -14706.139} C_VEL
LIN {X 0,Y 333.648,Z 494.051,A -85,B 0,C 180,E1 -14709.192,E2 -14709.192} C_VEL
LIN {X 0,Y 333.634,Z 494.048,A -85,B 0,C 180,E1 -14712.5,E2 -14712.5} C_VEL
LIN {X 0,Y 333.623,Z 494.05,A -85,B 0,C 180,E1 -14715.959,E2 -14715.959} C_VEL
LIN {X 0,Y 333.648,Z 494.052,A -85,B 0,C 180,E1 -14719.315,E2 -14719.315} C_VEL
LIN {X 0,Y 333.648,Z 494.049,A -85,B 0,C 180,E1 -14720.956,E2 -14720.956} C_VEL
LIN {X 0,Y 332.992,Z 494.137,A -85,B 0,C 180,E1 -14721.964,E2 -14721.964} C_VEL
LIN {X 0,Y 330.136,Z 494.494,A -85,B 0,C 180,E1 -14723.604,E2 -14723.604} C_VEL
LIN {X 0,Y 327.718,Z 494.792,A -85,B 0,C 180,E1 -14724.933,E2 -14724.933} C_VEL
LIN {X 0,Y 326.694,Z 494.916,A -85,B 0,C 180,E1 -14725.961,E2 -14725.961} C_VEL
LIN {X 0,Y 326.618,Z 494.924,A -85,B 0,C 180,E1 -14726.31,E2 -14726.31} C_VEL
LIN {X 0,Y 326.648,Z 495.002,A -85,B 0,C 180,E1 -14727.092,E2 -14727.092} C_VEL
LIN {X 0,Y 330.248,Z 510.708,A -85,B 0,C 180,E1 -14730.345,E2 -14730.345} C_VEL
LIN {X 0,Y 332.466,Z 521.886,A -85,B 0,C 180,E1 -14732.603,E2 -14732.603} C_VEL
LIN {X 0,Y 331.625,Z 534.456,A -85,B 0,C 180,E1 -14734.922,E2 -14734.922} C_VEL
LIN {X 0,Y 330.637,Z 549.006,A -85,B 0,C 180,E1 -14737.568,E2 -14737.568} C_VEL
LIN {X 0,Y 333.887,Z 576.061,A -85,B 0,C 180,E1 -14738.553,E2 -14738.553} C_VEL
LIN {X 0,Y 331.362,Z 660.03,A -85,B 0,C 180,E1 -14741.048,E2 -14741.048} C_VEL
LIN {X 0,Y 330.719,Z 673.166,A -85,B 0,C 180,E1 -14741.653,E2 -14741.653} C_VEL
LIN {X 0,Y 329.952,Z 687.019,A -85,B 0,C 180,E1 -14742.571,E2 -14742.571} C_VEL
LIN {X 0,Y 329.172,Z 698.49,A -85,B 0,C 180,E1 -14743.567,E2 -14743.567} C_VEL
LIN {X 0,Y 328.492,Z 708.857,A -85,B 0,C 180,E1 -14744.696,E2 -14744.696} C_VEL
LIN {X 0,Y 327.618,Z 720.037,A -85,B 0,C 180,E1 -14746.193,E2 -14746.193} C_VEL
LIN {X 0,Y 326.737,Z 730.168,A -85,B 0,C 180,E1 -14747.894,E2 -14747.894} C_VEL
LIN {X 0,Y 326.024,Z 739.104,A -85,B 0,C 180,E1 -14749.756,E2 -14749.756} C_VEL
LIN {X 0,Y 325.501,Z 746.208,A -85,B 0,C 180,E1 -14751.62,E2 -14751.62} C_VEL
LIN {X 0,Y 325.193,Z 752.726,A -85,B 0,C 180,E1 -14753.797,E2 -14753.797} C_VEL
LIN {X 0,Y 325.04,Z 756.913,A -85,B 0,C 180,E1 -14755.66,E2 -14755.66} C_VEL
LIN {X 0,Y 324.887,Z 759.972,A -85,B 0,C 180,E1 -14757.52,E2 -14757.52} C_VEL
LIN {X 0,Y 324.835,Z 761.417,A -85,B 0,C 180,E1 -14758.76,E2 -14758.76} C_VEL
LIN {X 0,Y 324.87,Z 762.444,A -85,B 0,C 180,E1 -14760,E2 -14760} C_VEL
LIN {X 0,Y 324.894,Z 763.003,A -85,B 0,C 180,E1 -14761.24,E2 -14761.24} C_VEL
LIN {X 0,Y 324.964,Z 763.112,A -85,B 0,C 180,E1 -14762.479,E2 -14762.479} C_VEL
LIN {X 0,Y 325.075,Z 762.807,A -85,B 0,C 180,E1 -14763.719,E2 -14763.719} C_VEL
LIN {X 0,Y 325.31,Z 762.059,A -85,B 0,C 180,E1 -14764.957,E2 -14764.957} C_VEL
LIN {X 0,Y 325.666,Z 760.845,A -85,B 0,C 180,E1 -14766.194,E2 -14766.194} C_VEL
LIN {X 0,Y 326.084,Z 758.227,A -85,B 0,C 180,E1 -14768.053,E2 -14768.053} C_VEL
LIN {X 0,Y 326.764,Z 754.531,A -85,B 0,C 180,E1 -14769.908,E2 -14769.908} C_VEL
LIN {X 0,Y 327.747,Z 749.668,A -85,B 0,C 180,E1 -14771.754,E2 -14771.754} C_VEL
LIN {X 0,Y 328.882,Z 743.574,A -85,B 0,C 180,E1 -14773.595,E2 -14773.595} C_VEL
LIN {X 0,Y 330.435,Z 735.917,A -85,B 0,C 180,E1 -14775.418,E2 -14775.418} C_VEL
LIN {X 0,Y 332.25,Z 726.393,A -85,B 0,C 180,E1 -14777.226,E2 -14777.226} C_VEL
LIN {X 0,Y 334.239,Z 715.461,A -85,B 0,C 180,E1 -14778.877,E2 -14778.877} C_VEL
LIN {X 0,Y 335.93,Z 704.689,A -85,B 0,C 180,E1 -14780.194,E2 -14780.194} C_VEL
LIN {X 0,Y 337.467,Z 694.188,A -85,B 0,C 180,E1 -14781.214,E2 -14781.214} C_VEL
LIN {X 0,Y 339.101,Z 680.963,A -85,B 0,C 180,E1 -14782.225,E2 -14782.225} C_VEL
LIN {X 0,Y 340.479,Z 667.774,A -85,B 0,C 180,E1 -14782.97,E2 -14782.97} C_VEL
LIN {X 0,Y 341.532,Z 653.521,A -85,B 0,C 180,E1 -14783.537,E2 -14783.537} C_VEL
LIN {X 0,Y 346.899,Z 584.455,A -85,B 0,C 180,E1 -14785.925,E2 -14785.925} C_VEL
LIN {X 0,Y 347.087,Z 580.224,A -85,B 0,C 180,E1 -14786.101,E2 -14786.101} C_VEL
LIN {X 0,Y 344.934,Z 566.187,A -85,B 0,C 180,E1 -14787.159,E2 -14787.159} C_VEL
LIN {X 0,Y 342.035,Z 551.873,A -85,B 0,C 180,E1 -14788.496,E2 -14788.496} C_VEL
LIN {X 0,Y 343.655,Z 542.431,A -85,B 0,C 180,E1 -14790.412,E2 -14790.412} C_VEL
LIN {X 0,Y 342.947,Z 536.005,A -85,B 0,C 180,E1 -14792.196,E2 -14792.196} C_VEL
LIN {X 0,Y 341.782,Z 529.941,A -85,B 0,C 180,E1 -14794.135,E2 -14794.135} C_VEL
LIN {X 0,Y 340.32,Z 524.176,A -85,B 0,C 180,E1 -14796.351,E2 -14796.351} C_VEL
LIN {X 0,Y 338.575,Z 518.663,A -85,B 0,C 180,E1 -14799.016,E2 -14799.016} C_VEL
LIN {X 0,Y 337.047,Z 514.473,A -85,B 0,C 180,E1 -14801.856,E2 -14801.856} C_VEL
LIN {X 0,Y 336.364,Z 512.816,A -85,B 0,C 180,E1 -14803.591,E2 -14803.591} C_VEL
LIN {X 0,Y 335.88,Z 511.553,A -85,B 0,C 180,E1 -14806.33,E2 -14806.33} C_VEL
LIN {X 0,Y 336.037,Z 511.493,A -85,B 0,C 180,E1 -14807.99,E2 -14807.99} C_VEL
LIN {X 0,Y 336.89,Z 512.713,A -85,B 0,C 180,E1 -14810.523,E2 -14810.523} C_VEL
LIN {X 0,Y 338.909,Z 515.177,A -85,B 0,C 180,E1 -14813.031,E2 -14813.031} C_VEL
LIN {X 0,Y 341.443,Z 519.498,A -85,B 0,C 180,E1 -14815.42,E2 -14815.42} C_VEL
LIN {X 0,Y 341.918,Z 520.599,A -85,B 0,C 180,E1 -14815.884,E2 -14815.884} C_VEL
LIN {X 0,Y 342.755,Z 525.802,A -85,B 0,C 180,E1 -14817.212,E2 -14817.212} C_VEL
LIN {X 0,Y 344.732,Z 535.715,A -85,B 0,C 180,E1 -14819.358,E2 -14819.358} C_VEL
LIN {X 0,Y 345.571,Z 540.897,A -85,B 0,C 180,E1 -14820.254,E2 -14820.254} C_VEL
LIN {X 0,Y 345.364,Z 546.822,A -85,B 0,C 180,E1 -14820.942,E2 -14820.942} C_VEL
LIN {X 0,Y 344.445,Z 559.545,A -85,B 0,C 180,E1 -14822.13,E2 -14822.13} C_VEL
LIN {X 0,Y 344.409,Z 563.613,A -85,B 0,C 180,E1 -14822.339,E2 -14822.339} C_VEL
LIN {X 0,Y 337.465,Z 653.744,A -85,B 0,C 180,E1 -14825.713,E2 -14825.713} C_VEL
LIN {X 0,Y 335.882,Z 680.15,A -85,B 0,C 180,E1 -14826.738,E2 -14826.738} C_VEL
LIN {X 0,Y 334.959,Z 693.311,A -85,B 0,C 180,E1 -14827.486,E2 -14827.486} C_VEL
LIN {X 0,Y 333.739,Z 706.822,A -85,B 0,C 180,E1 -14828.518,E2 -14828.518} C_VEL
LIN {X 0,Y 332.34,Z 719.243,A -85,B 0,C 180,E1 -14829.74,E2 -14829.74} C_VEL
LIN {X 0,Y 330.887,Z 730.402,A -85,B 0,C 180,E1 -14831.101,E2 -14831.101} C_VEL
LIN {X 0,Y 329.568,Z 740.548,A -85,B 0,C 180,E1 -14832.63,E2 -14832.63} C_VEL
LIN {X 0,Y 328.358,Z 749.105,A -85,B 0,C 180,E1 -14834.204,E2 -14834.204} C_VEL
LIN {X 0,Y 327.279,Z 757.258,A -85,B 0,C 180,E1 -14836.02,E2 -14836.02} C_VEL
LIN {X 0,Y 326.383,Z 764.023,A -85,B 0,C 180,E1 -14837.881,E2 -14837.881} C_VEL
LIN {X 0,Y 325.627,Z 770.18,A -85,B 0,C 180,E1 -14840.057,E2 -14840.057} C_VEL
LIN {X 0,Y 325.22,Z 774.203,A -85,B 0,C 180,E1 -14841.925,E2 -14841.925} C_VEL
LIN {X 0,Y 325.008,Z 777.543,A -85,B 0,C 180,E1 -14844.104,E2 -14844.104} C_VEL
LIN {X 0,Y 324.878,Z 779.491,A -85,B 0,C 180,E1 -14846.279,E2 -14846.279} C_VEL
LIN {X 0,Y 324.889,Z 780.093,A -85,B 0,C 180,E1 -14848.761,E2 -14848.761} C_VEL
LIN {X 0,Y 324.909,Z 780.775,A -85,B 0,C 180,E1 -14850,E2 -14850} C_VEL
LIN {X 0,Y 324.843,Z 781.011,A -85,B 0,C 180,E1 -14852.48,E2 -14852.48} C_VEL
LIN {X 0,Y 324.869,Z 780.573,A -85,B 0,C 180,E1 -14853.721,E2 -14853.721} C_VEL
LIN {X 0,Y 324.959,Z 778.596,A -85,B 0,C 180,E1 -14856.208,E2 -14856.208} C_VEL
LIN {X 0,Y 325.138,Z 777.053,A -85,B 0,C 180,E1 -14857.452,E2 -14857.452} C_VEL
LIN {X 0,Y 325.649,Z 772.778,A -85,B 0,C 180,E1 -14859.942,E2 -14859.942} C_VEL
LIN {X 0,Y 326.533,Z 766.854,A -85,B 0,C 180,E1 -14862.429,E2 -14862.429} C_VEL
LIN {X 0,Y 327.778,Z 760.182,A -85,B 0,C 180,E1 -14864.592,E2 -14864.592} C_VEL
LIN {X 0,Y 329.07,Z 753.21,A -85,B 0,C 180,E1 -14866.438,E2 -14866.438} C_VEL
LIN {X 0,Y 330.959,Z 743.35,A -85,B 0,C 180,E1 -14868.574,E2 -14868.574} C_VEL
LIN {X 0,Y 333.037,Z 732.983,A -85,B 0,C 180,E1 -14870.377,E2 -14870.377} C_VEL
LIN {X 0,Y 335.226,Z 721.522,A -85,B 0,C 180,E1 -14872.009,E2 -14872.009} C_VEL
LIN {X 0,Y 337.571,Z 708.626,A -85,B 0,C 180,E1 -14873.491,E2 -14873.491} C_VEL
LIN {X 0,Y 339.57,Z 696.434,A -85,B 0,C 180,E1 -14874.615,E2 -14874.615} C_VEL
LIN {X 0,Y 341.463,Z 682.788,A -85,B 0,C 180,E1 -14875.609,E2 -14875.609} C_VEL
LIN {X 0,Y 343.33,Z 667.315,A -85,B 0,C 180,E1 -14876.438,E2 -14876.438} C_VEL
LIN {X 0,Y 344.611,Z 651.586,A -85,B 0,C 180,E1 -14877.027,E2 -14877.027} C_VEL
LIN {X 0,Y 349.632,Z 587.426,A -85,B 0,C 180,E1 -14879.106,E2 -14879.106} C_VEL
LIN {X 0,Y 351.778,Z 562.235,A -85,B 0,C 180,E1 -14879.965,E2 -14879.965} C_VEL
LIN {X 0,Y 350.404,Z 550.69,A -85,B 0,C 180,E1 -14880.802,E2 -14880.802} C_VEL
LIN {X 0,Y 347.328,Z 544.388,A -85,B 0,C 180,E1 -14881.759,E2 -14881.759} C_VEL
LIN {X 0,Y 344.65,Z 539.713,A -85,B 0,C 180,E1 -14882.613,E2 -14882.613} C_VEL
LIN {X 0,Y 342.465,Z 535.924,A -85,B 0,C 180,E1 -14883.376,E2 -14883.376} C_VEL
LIN {X 0,Y 339.827,Z 531.481,A -85,B 0,C 180,E1 -14884.402,E2 -14884.402} C_VEL
LIN {X 0,Y 338.635,Z 526.942,A -85,B 0,C 180,E1 -14887.004,E2 -14887.004} C_VEL
LIN {X 0,Y 337.645,Z 523.684,A -85,B 0,C 180,E1 -14889.633,E2 -14889.633} C_VEL
LIN {X 0,Y 337.094,Z 521.783,A -85,B 0,C 180,E1 -14891.849,E2 -14891.849} C_VEL
LIN {X 0,Y 336.648,Z 520.669,A -85,B 0,C 180,E1 -14894.781,E2 -14894.781} C_VEL
LIN {X 0,Y 336.671,Z 520.752,A -85,B 0,C 180,E1 -14896.939,E2 -14896.939} C_VEL
LIN {X 0,Y 337.051,Z 521.971,A -85,B 0,C 180,E1 -14899.73,E2 -14899.73} C_VEL
LIN {X 0,Y 337.861,Z 524.969,A -85,B 0,C 180,E1 -14902.898,E2 -14902.898} C_VEL
LIN {X 0,Y 338.934,Z 529.422,A -85,B 0,C 180,E1 -14905.954,E2 -14905.954} C_VEL
LIN {X 0,Y 340.038,Z 535.267,A -85,B 0,C 180,E1 -14908.888,E2 -14908.888} C_VEL
LIN {X 0,Y 340.391,Z 537.229,A -85,B 0,C 180,E1 -14909.674,E2 -14909.674} C_VEL
LIN {X 0,Y 343.658,Z 543.703,A -85,B 0,C 180,E1 -14910.923,E2 -14910.923} C_VEL
LIN {X 0,Y 344.789,Z 546.754,A -85,B 0,C 180,E1 -14911.371,E2 -14911.371} C_VEL
LIN {X 0,Y 347.617,Z 560.813,A -85,B 0,C 180,E1 -14912.821,E2 -14912.821} C_VEL
LIN {X 0,Y 349.38,Z 572.398,A -85,B 0,C 180,E1 -14913.803,E2 -14913.803} C_VEL
LIN {X 0,Y 350.017,Z 579.589,A -85,B 0,C 180,E1 -14914.314,E2 -14914.314} C_VEL
LIN {X 0,Y 342.704,Z 659.289,A -85,B 0,C 180,E1 -14917.287,E2 -14917.287} C_VEL
LIN {X 0,Y 341.348,Z 671.678,A -85,B 0,C 180,E1 -14917.961,E2 -14917.961} C_VEL
LIN {X 0,Y 339.499,Z 685.041,A -85,B 0,C 180,E1 -14918.919,E2 -14918.919} C_VEL
LIN {X 0,Y 337.535,Z 697.985,A -85,B 0,C 180,E1 -14920.118,E2 -14920.118} C_VEL
LIN {X 0,Y 335.65,Z 708.924,A -85,B 0,C 180,E1 -14921.379,E2 -14921.379} C_VEL
LIN {X 0,Y 333.658,Z 719.345,A -85,B 0,C 180,E1 -14922.849,E2 -14922.849} C_VEL
LIN {X 0,Y 331.905,Z 727.992,A -85,B 0,C 180,E1 -14924.337,E2 -14924.337} C_VEL
LIN {X 0,Y 330.241,Z 736.632,A -85,B 0,C 180,E1 -14926.148,E2 -14926.148} C_VEL
LIN {X 0,Y 328.781,Z 743.614,A -85,B 0,C 180,E1 -14927.97,E2 -14927.97} C_VEL
LIN {X 0,Y 327.768,Z 748.411,A -85,B 0,C 180,E1 -14929.499,E2 -14929.499} C_VEL
LIN {X 0,Y 326.63,Z 753.999,A -85,B 0,C 180,E1 -14931.799,E2 -14931.799} C_VEL
LIN {X 0,Y 325.802,Z 757.519,A -85,B 0,C 180,E1 -14933.808,E2 -14933.808} C_VEL
LIN {X 0,Y 325.518,Z 759.085,A -85,B 0,C 180,E1 -14935.046,E2 -14935.046} C_VEL
LIN {X 0,Y 325.358,Z 760.195,A -85,B 0,C 180,E1 -14936.284,E2 -14936.284} C_VEL
LIN {X 0,Y 325.161,Z 760.863,A -85,B 0,C 180,E1 -14937.522,E2 -14937.522} C_VEL
LIN {X 0,Y 325.001,Z 761.123,A -85,B 0,C 180,E1 -14938.761,E2 -14938.761} C_VEL
LIN {X 0,Y 324.914,Z 760.965,A -85,B 0,C 180,E1 -14940,E2 -14940} C_VEL
LIN {X 0,Y 324.877,Z 760.355,A -85,B 0,C 180,E1 -14941.24,E2 -14941.24} C_VEL
LIN {X 0,Y 324.894,Z 759.29,A -85,B 0,C 180,E1 -14942.48,E2 -14942.48} C_VEL
LIN {X 0,Y 324.958,Z 757.799,A -85,B 0,C 180,E1 -14943.72,E2 -14943.72} C_VEL
LIN {X 0,Y 325.002,Z 754.891,A -85,B 0,C 180,E1 -14945.479,E2 -14945.479} C_VEL
LIN {X 0,Y 325.217,Z 750.469,A -85,B 0,C 180,E1 -14947.45,E2 -14947.45} C_VEL
LIN {X 0,Y 325.552,Z 745.028,A -85,B 0,C 180,E1 -14949.318,E2 -14949.318} C_VEL
LIN {X 0,Y 326.005,Z 738.203,A -85,B 0,C 180,E1 -14951.188,E2 -14951.188} C_VEL
LIN {X 0,Y 326.812,Z 729.669,A -85,B 0,C 180,E1 -14953.05,E2 -14953.05} C_VEL
LIN {X 0,Y 327.4,Z 720.983,A -85,B 0,C 180,E1 -14954.609,E2 -14954.609} C_VEL
LIN {X 0,Y 328.325,Z 710.505,A -85,B 0,C 180,E1 -14956.157,E2 -14956.157} C_VEL
LIN {X 0,Y 329.335,Z 698.822,A -85,B 0,C 180,E1 -14957.543,E2 -14957.543} C_VEL
LIN {X 0,Y 330.219,Z 687.643,A -85,B 0,C 180,E1 -14958.617,E2 -14958.617} C_VEL
LIN {X 0,Y 331.121,Z 674.507,A -85,B 0,C 180,E1 -14959.61,E2 -14959.61} C_VEL
LIN {X 0,Y 331.847,Z 660.054,A -85,B 0,C 180,E1 -14960.413,E2 -14960.413} C_VEL
LIN {X 0,Y 332.501,Z 645.816,A -85,B 0,C 180,E1 -14960.937,E2 -14960.937} C_VEL
LIN {X 0,Y 335.062,Z 572.934,A -85,B 0,C 180,E1 -14963.159,E2 -14963.159} C_VEL
LIN {X 0,Y 330.737,Z 539.152,A -85,B 0,C 180,E1 -14964.511,E2 -14964.511} C_VEL
LIN {X 0,Y 332.606,Z 523.459,A -85,B 0,C 180,E1 -14968.044,E2 -14968.044} C_VEL
LIN {X 0,Y 332.285,Z 520.488,A -85,B 0,C 180,E1 -14968.762,E2 -14968.762} C_VEL
LIN {X 0,Y 328.976,Z 505.41,A -85,B 0,C 180,E1 -14972.603,E2 -14972.603} C_VEL
LIN {X 0,Y 326.674,Z 494.919,A -85,B 0,C 180,E1 -14975.397,E2 -14975.397} C_VEL
LIN {X 0,Y 326.614,Z 494.925,A -85,B 0,C 180,E1 -14979.227,E2 -14979.227} C_VEL
LIN {X 0,Y 326.578,Z 494.928,A -85,B 0,C 180,E1 -14982.972,E2 -14982.972} C_VEL
LIN {X 0,Y 326.578,Z 494.928,A -85,B 0,C 180,E1 -14987.028,E2 -14987.028} C_VEL
LIN {X 0,Y 326.613,Z 494.923,A -85,B 0,C 180,E1 -14990.773,E2 -14990.773} C_VEL
LIN {X 0,Y 326.614,Z 494.922,A -85,B 0,C 180,E1 -14994.48,E2 -14994.48} C_VEL
LIN {X 0,Y 326.612,Z 494.928,A -85,B 0,C 180,E1 -14997.456,E2 -14997.456} C_VEL
LIN {X 0,Y 326.662,Z 494.916,A -85,B 0,C 180,E1 -15000.341,E2 -15000.341} C_VEL
LIN {X 0,Y 326.691,Z 494.913,A -85,B 0,C 180,E1 -15004.516,E2 -15004.516} C_VEL
LIN {X 0,Y 326.651,Z 494.918,A -85,B 0,C 180,E1 -15008.545,E2 -15008.545} C_VEL
LIN {X 0,Y 326.746,Z 494.909,A -85,B 0,C 180,E1 -15011.177,E2 -15011.177} C_VEL
LIN {X 0,Y 326.764,Z 494.909,A -85,B 0,C 180,E1 -15015.433,E2 -15015.433} C_VEL
LIN {X 0,Y 326.772,Z 494.903,A -85,B 0,C 180,E1 -15018.839,E2 -15018.839} C_VEL
LIN {X 0,Y 326.981,Z 494.877,A -85,B 0,C 180,E1 -15022.59,E2 -15022.59} C_VEL
LIN {X 0,Y 326.78,Z 494.904,A -85,B 0,C 180,E1 -15025.065,E2 -15025.065} C_VEL
LIN {X 0,Y 327.07,Z 494.871,A -85,B 0,C 180,E1 -15027.537,E2 -15027.537} C_VEL
LIN {X 0,Y 327.219,Z 494.848,A -85,B 0,C 180,E1 -15030,E2 -15030} C_VEL
LIN {X 0,Y 327.05,Z 494.868,A -85,B 0,C 180,E1 -15032.463,E2 -15032.463} C_VEL
LIN {X 0,Y 326.997,Z 494.875,A -85,B 0,C 180,E1 -15036.169,E2 -15036.169} C_VEL
LIN {X 0,Y 326.916,Z 494.885,A -85,B 0,C 180,E1 -15038.655,E2 -15038.655} C_VEL
LIN {X 0,Y 326.736,Z 494.907,A -85,B 0,C 180,E1 -15042.421,E2 -15042.421} C_VEL
LIN {X 0,Y 326.755,Z 494.906,A -85,B 0,C 180,E1 -15044.957,E2 -15044.957} C_VEL
LIN {X 0,Y 326.734,Z 494.909,A -85,B 0,C 180,E1 -15048.838,E2 -15048.838} C_VEL
LIN {X 0,Y 326.622,Z 494.922,A -85,B 0,C 180,E1 -15052.787,E2 -15052.787} C_VEL
LIN {X 0,Y 326.691,Z 494.917,A -85,B 0,C 180,E1 -15055.484,E2 -15055.484} C_VEL
LIN {X 0,Y 326.649,Z 494.921,A -85,B 0,C 180,E1 -15059.66,E2 -15059.66} C_VEL
LIN {X 0,Y 326.608,Z 494.924,A -85,B 0,C 180,E1 -15064.019,E2 -15064.019} C_VEL
LIN {X 0,Y 326.63,Z 494.925,A -85,B 0,C 180,E1 -15067.239,E2 -15067.239} C_VEL
LIN {X 0,Y 326.579,Z 494.931,A -85,B 0,C 180,E1 -15071.132,E2 -15071.132} C_VEL
LIN {X 0,Y 326.557,Z 494.93,A -85,B 0,C 180,E1 -15074.748,E2 -15074.748} C_VEL
LIN {X 0,Y 326.578,Z 494.927,A -85,B 0,C 180,E1 -15078.154,E2 -15078.154} C_VEL
LIN {X 0,Y 326.625,Z 494.926,A -85,B 0,C 180,E1 -15081.392,E2 -15081.392} C_VEL
LIN {X 0,Y 326.621,Z 494.923,A -85,B 0,C 180,E1 -15084.851,E2 -15084.851} C_VEL
LIN {X 0,Y 326.618,Z 494.924,A -85,B 0,C 180,E1 -15086.31,E2 -15086.31} C_VEL
LIN {X 0,Y 326.481,Z 495.611,A -85,B 0,C 180,E1 -15086.905,E2 -15086.905} C_VEL
LIN {X 0,Y 326.003,Z 497.88,A -85,B 0,C 180,E1 -15087.587,E2 -15087.587} C_VEL
LIN {X 0,Y 323.615,Z 510.515,A -85,B 0,C 180,E1 -15089.883,E2 -15089.883} C_VEL
LIN {X 0,Y 323.846,Z 514.42,A -85,B 0,C 180,E1 -15090.66,E2 -15090.66} C_VEL
LIN {X 0,Y 325.458,Z 522.439,A -85,B 0,C 180,E1 -15092.296,E2 -15092.296} C_VEL
LIN {X 0,Y 325.408,Z 526.286,A -85,B 0,C 180,E1 -15093.028,E2 -15093.028} C_VEL
LIN {X 0,Y 323.823,Z 547.646,A -85,B 0,C 180,E1 -15097.005,E2 -15097.005} C_VEL
LIN {X 0,Y 323.713,Z 549.018,A -85,B 0,C 180,E1 -15097.252,E2 -15097.252} C_VEL
LIN {X 0,Y 326.967,Z 576.981,A -85,B 0,C 180,E1 -15098.293,E2 -15098.293} C_VEL
LIN {X 0,Y 324.303,Z 660.697,A -85,B 0,C 180,E1 -15100.866,E2 -15100.866} C_VEL
LIN {X 0,Y 323.688,Z 673.568,A -85,B 0,C 180,E1 -15101.486,E2 -15101.486} C_VEL
LIN {X 0,Y 322.923,Z 687.303,A -85,B 0,C 180,E1 -15102.424,E2 -15102.424} C_VEL
LIN {X 0,Y 322.055,Z 699.459,A -85,B 0,C 180,E1 -15103.519,E2 -15103.519} C_VEL
LIN {X 0,Y 321.302,Z 710.549,A -85,B 0,C 180,E1 -15104.783,E2 -15104.783} C_VEL
LIN {X 0,Y 320.499,Z 720.719,A -85,B 0,C 180,E1 -15106.204,E2 -15106.204} C_VEL
LIN {X 0,Y 319.605,Z 730.758,A -85,B 0,C 180,E1 -15107.942,E2 -15107.942} C_VEL
LIN {X 0,Y 319.018,Z 738.277,A -85,B 0,C 180,E1 -15109.528,E2 -15109.528} C_VEL
LIN {X 0,Y 318.459,Z 745.634,A -85,B 0,C 180,E1 -15111.433,E2 -15111.433} C_VEL
LIN {X 0,Y 318.126,Z 752.329,A -85,B 0,C 180,E1 -15113.658,E2 -15113.658} C_VEL
LIN {X 0,Y 317.958,Z 756.694,A -85,B 0,C 180,E1 -15115.563,E2 -15115.563} C_VEL
LIN {X 0,Y 317.809,Z 759.9,A -85,B 0,C 180,E1 -15117.465,E2 -15117.465} C_VEL
LIN {X 0,Y 317.747,Z 761.423,A -85,B 0,C 180,E1 -15118.733,E2 -15118.733} C_VEL
LIN {X 0,Y 317.778,Z 762.504,A -85,B 0,C 180,E1 -15120,E2 -15120} C_VEL
LIN {X 0,Y 317.805,Z 763.17,A -85,B 0,C 180,E1 -15121.267,E2 -15121.267} C_VEL
LIN {X 0,Y 317.883,Z 763.359,A -85,B 0,C 180,E1 -15122.534,E2 -15122.534} C_VEL
LIN {X 0,Y 318.012,Z 763.119,A -85,B 0,C 180,E1 -15123.801,E2 -15123.801} C_VEL
LIN {X 0,Y 318.27,Z 762.464,A -85,B 0,C 180,E1 -15125.067,E2 -15125.067} C_VEL
LIN {X 0,Y 318.831,Z 760.222,A -85,B 0,C 180,E1 -15127.28,E2 -15127.28} C_VEL
LIN {X 0,Y 319.53,Z 756.601,A -85,B 0,C 180,E1 -15129.495,E2 -15129.495} C_VEL
LIN {X 0,Y 320.517,Z 752.316,A -85,B 0,C 180,E1 -15131.382,E2 -15131.382} C_VEL
LIN {X 0,Y 321.623,Z 746.821,A -85,B 0,C 180,E1 -15133.264,E2 -15133.264} C_VEL
LIN {X 0,Y 323.13,Z 739.893,A -85,B 0,C 180,E1 -15135.129,E2 -15135.129} C_VEL
LIN {X 0,Y 324.993,Z 731.355,A -85,B 0,C 180,E1 -15136.974,E2 -15136.974} C_VEL
LIN {X 0,Y 326.862,Z 722.267,A -85,B 0,C 180,E1 -15138.558,E2 -15138.558} C_VEL
LIN {X 0,Y 328.77,Z 711.995,A -85,B 0,C 180,E1 -15140,E2 -15140} C_VEL
LIN {X 0,Y 330.592,Z 700.319,A -85,B 0,C 180,E1 -15141.35,E2 -15141.35} C_VEL
LIN {X 0,Y 332.607,Z 686.973,A -85,B 0,C 180,E1 -15142.519,E2 -15142.519} C_VEL
LIN {X 0,Y 334.176,Z 673.858,A -85,B 0,C 180,E1 -15143.388,E2 -15143.388} C_VEL
LIN {X 0,Y 335.494,Z 659.4,A -85,B 0,C 180,E1 -15144.069,E2 -15144.069} C_VEL
LIN {X 0,Y 341.962,Z 582.592,A -85,B 0,C 180,E1 -15146.815,E2 -15146.815} C_VEL
LIN {X 0,Y 340.045,Z 568.835,A -85,B 0,C 180,E1 -15147.897,E2 -15147.897} C_VEL
LIN {X 0,Y 337.106,Z 553.951,A -85,B 0,C 180,E1 -15149.348,E2 -15149.348} C_VEL
LIN {X 0,Y 336.858,Z 552.03,A -85,B 0,C 180,E1 -15149.583,E2 -15149.583} C_VEL
LIN {X 0,Y 338.059,Z 545.31,A -85,B 0,C 180,E1 -15151.015,E2 -15151.015} C_VEL
LIN {X 0,Y 337.369,Z 539.268,A -85,B 0,C 180,E1 -15152.795,E2 -15152.795} C_VEL
LIN {X 0,Y 336.283,Z 533.352,A -85,B 0,C 180,E1 -15154.827,E2 -15154.827} C_VEL
LIN {X 0,Y 334.954,Z 527.827,A -85,B 0,C 180,E1 -15157.125,E2 -15157.125} C_VEL
LIN {X 0,Y 333.581,Z 523.014,A -85,B 0,C 180,E1 -15159.715,E2 -15159.715} C_VEL
LIN {X 0,Y 332.38,Z 519.324,A -85,B 0,C 180,E1 -15162.58,E2 -15162.58} C_VEL
LIN {X 0,Y 331.942,Z 518.114,A -85,B 0,C 180,E1 -15164.322,E2 -15164.322} C_VEL
LIN {X 0,Y 331.746,Z 517.408,A -85,B 0,C 180,E1 -15166.078,E2 -15166.078} C_VEL
LIN {X 0,Y 332.019,Z 517.35,A -85,B 0,C 180,E1 -15167.805,E2 -15167.805} C_VEL
LIN {X 0,Y 332.533,Z 517.995,A -85,B 0,C 180,E1 -15169.539,E2 -15169.539} C_VEL
LIN {X 0,Y 334.506,Z 520.491,A -85,B 0,C 180,E1 -15172.461,E2 -15172.461} C_VEL
LIN {X 0,Y 336.076,Z 523.211,A -85,B 0,C 180,E1 -15174.159,E2 -15174.159} C_VEL
LIN {X 0,Y 337.426,Z 525.323,A -85,B 0,C 180,E1 -15175.279,E2 -15175.279} C_VEL
LIN {X 0,Y 337.89,Z 526.934,A -85,B 0,C 180,E1 -15175.834,E2 -15175.834} C_VEL
LIN {X 0,Y 339.336,Z 536.592,A -85,B 0,C 180,E1 -15178.12,E2 -15178.12} C_VEL
LIN {X 0,Y 340.592,Z 543.259,A -85,B 0,C 180,E1 -15179.44,E2 -15179.44} C_VEL
LIN {X 0,Y 340.471,Z 548.403,A -85,B 0,C 180,E1 -15180.108,E2 -15180.108} C_VEL
LIN {X 0,Y 339.459,Z 558.933,A -85,B 0,C 180,E1 -15181.137,E2 -15181.137} C_VEL
LIN {X 0,Y 339.612,Z 563.842,A -85,B 0,C 180,E1 -15181.457,E2 -15181.457} C_VEL
LIN {X 0,Y 332.502,Z 647.644,A -85,B 0,C 180,E1 -15184.7,E2 -15184.7} C_VEL
LIN {X 0,Y 330.224,Z 679.939,A -85,B 0,C 180,E1 -15185.982,E2 -15185.982} C_VEL
LIN {X 0,Y 329.192,Z 692.943,A -85,B 0,C 180,E1 -15186.734,E2 -15186.734} C_VEL
LIN {X 0,Y 327.955,Z 705.134,A -85,B 0,C 180,E1 -15187.678,E2 -15187.678} C_VEL
LIN {X 0,Y 326.512,Z 717.326,A -85,B 0,C 180,E1 -15188.867,E2 -15188.867} C_VEL
LIN {X 0,Y 324.814,Z 728.718,A -85,B 0,C 180,E1 -15190.24,E2 -15190.24} C_VEL
LIN {X 0,Y 323.407,Z 738.086,A -85,B 0,C 180,E1 -15191.633,E2 -15191.633} C_VEL
LIN {X 0,Y 322.053,Z 746.853,A -85,B 0,C 180,E1 -15193.193,E2 -15193.193} C_VEL
LIN {X 0,Y 320.805,Z 755.469,A -85,B 0,C 180,E1 -15195.083,E2 -15195.083} C_VEL
LIN {X 0,Y 319.584,Z 763.536,A -85,B 0,C 180,E1 -15197.296,E2 -15197.296} C_VEL
LIN {X 0,Y 318.828,Z 768.992,A -85,B 0,C 180,E1 -15199.201,E2 -15199.201} C_VEL
LIN {X 0,Y 318.308,Z 773.231,A -85,B 0,C 180,E1 -15201.109,E2 -15201.109} C_VEL
LIN {X 0,Y 318.056,Z 775.427,A -85,B 0,C 180,E1 -15202.381,E2 -15202.381} C_VEL
LIN {X 0,Y 317.892,Z 777.803,A -85,B 0,C 180,E1 -15204.192,E2 -15204.192} C_VEL
LIN {X 0,Y 317.788,Z 779.367,A -85,B 0,C 180,E1 -15206.196,E2 -15206.196} C_VEL
LIN {X 0,Y 317.786,Z 779.787,A -85,B 0,C 180,E1 -15207.465,E2 -15207.465} C_VEL
LIN {X 0,Y 317.797,Z 779.78,A -85,B 0,C 180,E1 -15208.733,E2 -15208.733} C_VEL
LIN {X 0,Y 317.762,Z 780.8,A -85,B 0,C 180,E1 -15211.267,E2 -15211.267} C_VEL
LIN {X 0,Y 317.778,Z 780.404,A -85,B 0,C 180,E1 -15213.804,E2 -15213.804} C_VEL
LIN {X 0,Y 317.888,Z 778.54,A -85,B 0,C 180,E1 -15216.347,E2 -15216.347} C_VEL
LIN {X 0,Y 318.29,Z 775.198,A -85,B 0,C 180,E1 -15218.892,E2 -15218.892} C_VEL
LIN {X 0,Y 318.806,Z 771.642,A -85,B 0,C 180,E1 -15220.8,E2 -15220.8} C_VEL
LIN {X 0,Y 319.998,Z 765.477,A -85,B 0,C 180,E1 -15223.333,E2 -15223.333} C_VEL
LIN {X 0,Y 321.148,Z 758.858,A -85,B 0,C 180,E1 -15225.463,E2 -15225.463} C_VEL
LIN {X 0,Y 322.819,Z 751.329,A -85,B 0,C 180,E1 -15227.419,E2 -15227.419} C_VEL
LIN {X 0,Y 324.652,Z 742.686,A -85,B 0,C 180,E1 -15229.277,E2 -15229.277} C_VEL
LIN {X 0,Y 326.886,Z 732.261,A -85,B 0,C 180,E1 -15231.108,E2 -15231.108} C_VEL
LIN {X 0,Y 329.202,Z 720.781,A -85,B 0,C 180,E1 -15232.765,E2 -15232.765} C_VEL
LIN {X 0,Y 331.752,Z 707.986,A -85,B 0,C 180,E1 -15234.245,E2 -15234.245} C_VEL
LIN {X 0,Y 333.901,Z 695.577,A -85,B 0,C 180,E1 -15235.395,E2 -15235.395} C_VEL
LIN {X 0,Y 335.937,Z 681.926,A -85,B 0,C 180,E1 -15236.396,E2 -15236.396} C_VEL
LIN {X 0,Y 337.907,Z 666.482,A -85,B 0,C 180,E1 -15237.231,E2 -15237.231} C_VEL
LIN {X 0,Y 339.405,Z 648.711,A -85,B 0,C 180,E1 -15237.895,E2 -15237.895} C_VEL
LIN {X 0,Y 345.029,Z 583.709,A -85,B 0,C 180,E1 -15240.074,E2 -15240.074} C_VEL
LIN {X 0,Y 346.88,Z 563.386,A -85,B 0,C 180,E1 -15240.8,E2 -15240.8} C_VEL
LIN {X 0,Y 345.758,Z 554.029,A -85,B 0,C 180,E1 -15241.533,E2 -15241.533} C_VEL
LIN {X 0,Y 341.904,Z 546.377,A -85,B 0,C 180,E1 -15242.837,E2 -15242.837} C_VEL
LIN {X 0,Y 338.84,Z 541.166,A -85,B 0,C 180,E1 -15243.937,E2 -15243.937} C_VEL
LIN {X 0,Y 336.107,Z 536.753,A -85,B 0,C 180,E1 -15245.02,E2 -15245.02} C_VEL
LIN {X 0,Y 333.13,Z 532.069,A -85,B 0,C 180,E1 -15246.395,E2 -15246.395} C_VEL
LIN {X 0,Y 332.293,Z 529.136,A -85,B 0,C 180,E1 -15248.505,E2 -15248.505} C_VEL
LIN {X 0,Y 331.562,Z 526.613,A -85,B 0,C 180,E1 -15251.079,E2 -15251.079} C_VEL
LIN {X 0,Y 331.078,Z 525.175,A -85,B 0,C 180,E1 -15253.802,E2 -15253.802} C_VEL
LIN {X 0,Y 330.966,Z 524.897,A -85,B 0,C 180,E1 -15256.219,E2 -15256.219} C_VEL
LIN {X 0,Y 331.206,Z 525.693,A -85,B 0,C 180,E1 -15258.868,E2 -15258.868} C_VEL
LIN {X 0,Y 331.693,Z 527.767,A -85,B 0,C 180,E1 -15261.626,E2 -15261.626} C_VEL
LIN {X 0,Y 332.555,Z 531.138,A -85,B 0,C 180,E1 -15264.467,E2 -15264.467} C_VEL
LIN {X 0,Y 333.302,Z 534.901,A -85,B 0,C 180,E1 -15266.754,E2 -15266.754} C_VEL
LIN {X 0,Y 333.728,Z 536.892,A -85,B 0,C 180,E1 -15267.718,E2 -15267.718} C_VEL
LIN {X 0,Y 337.391,Z 543.696,A -85,B 0,C 180,E1 -15269.358,E2 -15269.358} C_VEL
LIN {X 0,Y 339.96,Z 548.881,A -85,B 0,C 180,E1 -15270.388,E2 -15270.388} C_VEL
LIN {X 0,Y 340.742,Z 551.456,A -85,B 0,C 180,E1 -15270.76,E2 -15270.76} C_VEL
LIN {X 0,Y 343.101,Z 564.284,A -85,B 0,C 180,E1 -15272.121,E2 -15272.121} C_VEL
LIN {X 0,Y 344.558,Z 575.454,A -85,B 0,C 180,E1 -15273.097,E2 -15273.097} C_VEL
LIN {X 0,Y 344.952,Z 581.675,A -85,B 0,C 180,E1 -15273.528,E2 -15273.528} C_VEL
LIN {X 0,Y 337.247,Z 659.286,A -85,B 0,C 180,E1 -15276.515,E2 -15276.515} C_VEL
LIN {X 0,Y 335.72,Z 671.838,A -85,B 0,C 180,E1 -15277.215,E2 -15277.215} C_VEL
LIN {X 0,Y 333.729,Z 685.463,A -85,B 0,C 180,E1 -15278.212,E2 -15278.212} C_VEL
LIN {X 0,Y 331.745,Z 697.847,A -85,B 0,C 180,E1 -15279.378,E2 -15279.378} C_VEL
LIN {X 0,Y 329.59,Z 709.128,A -85,B 0,C 180,E1 -15280.7,E2 -15280.7} C_VEL
LIN {X 0,Y 327.482,Z 719.497,A -85,B 0,C 180,E1 -15282.193,E2 -15282.193} C_VEL
LIN {X 0,Y 325.602,Z 728.187,A -85,B 0,C 180,E1 -15283.704,E2 -15283.704} C_VEL
LIN {X 0,Y 323.739,Z 736.776,A -85,B 0,C 180,E1 -15285.543,E2 -15285.543} C_VEL
LIN {X 0,Y 321.946,Z 744.775,A -85,B 0,C 180,E1 -15287.711,E2 -15287.711} C_VEL
LIN {X 0,Y 320.861,Z 749.415,A -85,B 0,C 180,E1 -15289.27,E2 -15289.27} C_VEL
LIN {X 0,Y 319.881,Z 753.869,A -85,B 0,C 180,E1 -15291.153,E2 -15291.153} C_VEL
LIN {X 0,Y 319.344,Z 756.221,A -85,B 0,C 180,E1 -15292.412,E2 -15292.412} C_VEL
LIN {X 0,Y 318.787,Z 758.156,A -85,B 0,C 180,E1 -15293.671,E2 -15293.671} C_VEL
LIN {X 0,Y 318.465,Z 759.62,A -85,B 0,C 180,E1 -15294.936,E2 -15294.936} C_VEL
LIN {X 0,Y 318.28,Z 760.625,A -85,B 0,C 180,E1 -15296.202,E2 -15296.202} C_VEL
LIN {X 0,Y 318.076,Z 761.222,A -85,B 0,C 180,E1 -15297.467,E2 -15297.467} C_VEL
LIN {X 0,Y 317.909,Z 761.407,A -85,B 0,C 180,E1 -15298.733,E2 -15298.733} C_VEL
LIN {X 0,Y 317.82,Z 761.147,A -85,B 0,C 180,E1 -15300,E2 -15300} C_VEL
LIN {X 0,Y 317.787,Z 760.432,A -85,B 0,C 180,E1 -15301.267,E2 -15301.267} C_VEL
LIN {X 0,Y 317.813,Z 759.297,A -85,B 0,C 180,E1 -15302.535,E2 -15302.535} C_VEL
LIN {X 0,Y 317.856,Z 756.745,A -85,B 0,C 180,E1 -15304.438,E2 -15304.438} C_VEL
LIN {X 0,Y 318.026,Z 753.126,A -85,B 0,C 180,E1 -15306.344,E2 -15306.344} C_VEL
LIN {X 0,Y 318.245,Z 748.34,A -85,B 0,C 180,E1 -15308.253,E2 -15308.253} C_VEL
LIN {X 0,Y 318.658,Z 742.265,A -85,B 0,C 180,E1 -15310.162,E2 -15310.162} C_VEL
LIN {X 0,Y 319.233,Z 734.692,A -85,B 0,C 180,E1 -15312.072,E2 -15312.072} C_VEL
LIN {X 0,Y 320.066,Z 725.277,A -85,B 0,C 180,E1 -15313.977,E2 -15313.977} C_VEL
LIN {X 0,Y 320.818,Z 715.688,A -85,B 0,C 180,E1 -15315.566,E2 -15315.566} C_VEL
LIN {X 0,Y 321.795,Z 705.213,A -85,B 0,C 180,E1 -15316.984,E2 -15316.984} C_VEL
LIN {X 0,Y 322.897,Z 692.243,A -85,B 0,C 180,E1 -15318.397,E2 -15318.397} C_VEL
LIN {X 0,Y 323.802,Z 679.324,A -85,B 0,C 180,E1 -15319.494,E2 -15319.494} C_VEL
LIN {X 0,Y 324.621,Z 666.001,A -85,B 0,C 180,E1 -15320.35,E2 -15320.35} C_VEL
LIN {X 0,Y 325.332,Z 652.533,A -85,B 0,C 180,E1 -15320.965,E2 -15320.965} C_VEL
LIN {X 0,Y 328.191,Z 573.708,A -85,B 0,C 180,E1 -15323.454,E2 -15323.454} C_VEL
LIN {X 0,Y 323.885,Z 539.592,A -85,B 0,C 180,E1 -15324.829,E2 -15324.829} C_VEL
LIN {X 0,Y 323.933,Z 538.699,A -85,B 0,C 180,E1 -15324.96,E2 -15324.96} C_VEL
LIN {X 0,Y 325.668,Z 523.973,A -85,B 0,C 180,E1 -15328.344,E2 -15328.344} C_VEL
LIN {X 0,Y 323.483,Z 513.347,A -85,B 0,C 180,E1 -15331.063,E2 -15331.063} C_VEL
LIN {X 0,Y 320.415,Z 499.404,A -85,B 0,C 180,E1 -15334.77,E2 -15334.77} C_VEL
LIN {X 0,Y 319.636,Z 495.796,A -85,B 0,C 180,E1 -15335.812,E2 -15335.812} C_VEL
LIN {X 0,Y 319.56,Z 495.806,A -85,B 0,C 180,E1 -15339.668,E2 -15339.668} C_VEL
LIN {X 0,Y 319.523,Z 495.81,A -85,B 0,C 180,E1 -15343.46,E2 -15343.46} C_VEL
LIN {X 0,Y 319.556,Z 495.803,A -85,B 0,C 180,E1 -15347.016,E2 -15347.016} C_VEL
LIN {X 0,Y 319.548,Z 495.803,A -85,B 0,C 180,E1 -15350.371,E2 -15350.371} C_VEL
LIN {X 0,Y 319.56,Z 495.807,A -85,B 0,C 180,E1 -15353.572,E2 -15353.572} C_VEL
LIN {X 0,Y 319.579,Z 495.799,A -85,B 0,C 180,E1 -15356.686,E2 -15356.686} C_VEL
LIN {X 0,Y 319.593,Z 495.802,A -85,B 0,C 180,E1 -15359.617,E2 -15359.617} C_VEL
LIN {X 0,Y 319.61,Z 495.795,A -85,B 0,C 180,E1 -15362.498,E2 -15362.498} C_VEL
LIN {X 0,Y 319.607,Z 495.799,A -85,B 0,C 180,E1 -15365.304,E2 -15365.304} C_VEL
LIN {X 0,Y 319.599,Z 495.797,A -85,B 0,C 180,E1 -15368.048,E2 -15368.048} C_VEL
LIN {X 0,Y 319.691,Z 495.786,A -85,B 0,C 180,E1 -15370.962,E2 -15370.962} C_VEL
LIN {X 0,Y 319.732,Z 495.783,A -85,B 0,C 180,E1 -15375.276,E2 -15375.276} C_VEL
LIN {X 0,Y 319.759,Z 495.778,A -85,B 0,C 180,E1 -15379.873,E2 -15379.873} C_VEL
LIN {X 0,Y 319.935,Z 495.754,A -85,B 0,C 180,E1 -15382.426,E2 -15382.426} C_VEL
LIN {X 0,Y 319.75,Z 495.779,A -85,B 0,C 180,E1 -15384.956,E2 -15384.956} C_VEL
LIN {X 0,Y 320.01,Z 495.751,A -85,B 0,C 180,E1 -15387.482,E2 -15387.482} C_VEL
LIN {X 0,Y 320.17,Z 495.726,A -85,B 0,C 180,E1 -15390,E2 -15390} C_VEL
LIN {X 0,Y 319.994,Z 495.747,A -85,B 0,C 180,E1 -15392.518,E2 -15392.518} C_VEL
LIN {X 0,Y 319.953,Z 495.752,A -85,B 0,C 180,E1 -15396.305,E2 -15396.305} C_VEL
LIN {X 0,Y 319.844,Z 495.767,A -85,B 0,C 180,E1 -15398.848,E2 -15398.848} C_VEL
LIN {X 0,Y 319.683,Z 495.786,A -85,B 0,C 180,E1 -15402.7,E2 -15402.7} C_VEL
LIN {X 0,Y 319.701,Z 495.788,A -85,B 0,C 180,E1 -15405.295,E2 -15405.295} C_VEL
LIN {X 0,Y 319.676,Z 495.791,A -85,B 0,C 180,E1 -15409.255,E2 -15409.255} C_VEL
LIN {X 0,Y 319.572,Z 495.805,A -85,B 0,C 180,E1 -15413.319,E2 -15413.319} C_VEL
LIN {X 0,Y 319.619,Z 495.794,A -85,B 0,C 180,E1 -15416.089,E2 -15416.089} C_VEL
LIN {X 0,Y 319.581,Z 495.8,A -85,B 0,C 180,E1 -15418.935,E2 -15418.935} C_VEL
LIN {X 0,Y 319.531,Z 495.806,A -85,B 0,C 180,E1 -15421.862,E2 -15421.862} C_VEL
LIN {X 0,Y 319.582,Z 495.802,A -85,B 0,C 180,E1 -15425.543,E2 -15425.543} C_VEL
LIN {X 0,Y 319.575,Z 495.8,A -85,B 0,C 180,E1 -15428.008,E2 -15428.008} C_VEL
LIN {X 0,Y 319.527,Z 495.808,A -85,B 0,C 180,E1 -15431.597,E2 -15431.597} C_VEL
LIN {X 0,Y 319.517,Z 495.812,A -85,B 0,C 180,E1 -15435.262,E2 -15435.262} C_VEL
LIN {X 0,Y 319.529,Z 495.806,A -85,B 0,C 180,E1 -15438.712,E2 -15438.712} C_VEL
LIN {X 0,Y 319.563,Z 495.801,A -85,B 0,C 180,E1 -15442.348,E2 -15442.348} C_VEL
LIN {X 0,Y 319.564,Z 495.805,A -85,B 0,C 180,E1 -15445.124,E2 -15445.124} C_VEL
LIN {X 0,Y 319.628,Z 495.872,A -85,B 0,C 180,E1 -15446.761,E2 -15446.761} C_VEL
LIN {X 0,Y 323.096,Z 511.138,A -85,B 0,C 180,E1 -15449.98,E2 -15449.98} C_VEL
LIN {X 0,Y 323.846,Z 514.42,A -85,B 0,C 180,E1 -15450.66,E2 -15450.66} C_VEL
LIN {X 0,Y 323.831,Z 518.423,A -85,B 0,C 180,E1 -15451.426,E2 -15451.426} C_VEL
LIN {X 0,Y 322.657,Z 522.584,A -85,B 0,C 180,E1 -15452.153,E2 -15452.153} C_VEL
LIN {X 0,Y 318.208,Z 533.824,A -85,B 0,C 180,E1 -15454.069,E2 -15454.069} C_VEL
LIN {X 0,Y 317.727,Z 536.622,A -85,B 0,C 180,E1 -15454.586,E2 -15454.586} C_VEL
LIN {X 0,Y 316.818,Z 549.236,A -85,B 0,C 180,E1 -15456.942,E2 -15456.942} C_VEL
LIN {X 0,Y 320.086,Z 576.779,A -85,B 0,C 180,E1 -15457.998,E2 -15457.998} C_VEL
LIN {X 0,Y 317.295,Z 660.793,A -85,B 0,C 180,E1 -15460.679,E2 -15460.679} C_VEL
LIN {X 0,Y 316.657,Z 673.647,A -85,B 0,C 180,E1 -15461.311,E2 -15461.311} C_VEL
LIN {X 0,Y 315.881,Z 687.388,A -85,B 0,C 180,E1 -15462.27,E2 -15462.27} C_VEL
LIN {X 0,Y 315.013,Z 699.605,A -85,B 0,C 180,E1 -15463.394,E2 -15463.394} C_VEL
LIN {X 0,Y 314.287,Z 710.05,A -85,B 0,C 180,E1 -15464.601,E2 -15464.601} C_VEL
LIN {X 0,Y 313.462,Z 720.359,A -85,B 0,C 180,E1 -15466.053,E2 -15466.053} C_VEL
LIN {X 0,Y 312.622,Z 729.689,A -85,B 0,C 180,E1 -15467.669,E2 -15467.669} C_VEL
LIN {X 0,Y 311.885,Z 738.827,A -85,B 0,C 180,E1 -15469.614,E2 -15469.614} C_VEL
LIN {X 0,Y 311.33,Z 746.112,A -85,B 0,C 180,E1 -15471.562,E2 -15471.562} C_VEL
LIN {X 0,Y 311.043,Z 751.906,A -85,B 0,C 180,E1 -15473.513,E2 -15473.513} C_VEL
LIN {X 0,Y 310.878,Z 756.404,A -85,B 0,C 180,E1 -15475.462,E2 -15475.462} C_VEL
LIN {X 0,Y 310.735,Z 759.743,A -85,B 0,C 180,E1 -15477.407,E2 -15477.407} C_VEL
LIN {X 0,Y 310.663,Z 761.394,A -85,B 0,C 180,E1 -15478.704,E2 -15478.704} C_VEL
LIN {X 0,Y 310.688,Z 762.548,A -85,B 0,C 180,E1 -15480,E2 -15480} C_VEL
LIN {X 0,Y 310.718,Z 763.287,A -85,B 0,C 180,E1 -15481.296,E2 -15481.296} C_VEL
LIN {X 0,Y 310.805,Z 763.601,A -85,B 0,C 180,E1 -15482.592,E2 -15482.592} C_VEL
LIN {X 0,Y 310.952,Z 763.432,A -85,B 0,C 180,E1 -15483.888,E2 -15483.888} C_VEL
LIN {X 0,Y 311.232,Z 762.841,A -85,B 0,C 180,E1 -15485.182,E2 -15485.182} C_VEL
LIN {X 0,Y 311.796,Z 760.902,A -85,B 0,C 180,E1 -15487.351,E2 -15487.351} C_VEL
LIN {X 0,Y 312.585,Z 757.349,A -85,B 0,C 180,E1 -15489.708,E2 -15489.708} C_VEL
LIN {X 0,Y 313.619,Z 753.202,A -85,B 0,C 180,E1 -15491.636,E2 -15491.636} C_VEL
LIN {X 0,Y 315.021,Z 746.907,A -85,B 0,C 180,E1 -15493.876,E2 -15493.876} C_VEL
LIN {X 0,Y 316.735,Z 739.985,A -85,B 0,C 180,E1 -15495.772,E2 -15495.772} C_VEL
LIN {X 0,Y 318.737,Z 731.377,A -85,B 0,C 180,E1 -15497.649,E2 -15497.649} C_VEL
LIN {X 0,Y 320.837,Z 721.719,A -85,B 0,C 180,E1 -15499.347,E2 -15499.347} C_VEL
LIN {X 0,Y 322.989,Z 710.919,A -85,B 0,C 180,E1 -15500.874,E2 -15500.874} C_VEL
LIN {X 0,Y 324.776,Z 700.392,A -85,B 0,C 180,E1 -15502.085,E2 -15502.085} C_VEL
LIN {X 0,Y 326.911,Z 687.031,A -85,B 0,C 180,E1 -15503.268,E2 -15503.268} C_VEL
LIN {X 0,Y 328.582,Z 674.132,A -85,B 0,C 180,E1 -15504.146,E2 -15504.146} C_VEL
LIN {X 0,Y 330,Z 660.11,A -85,B 0,C 180,E1 -15504.831,E2 -15504.831} C_VEL
LIN {X 0,Y 336.788,Z 585.422,A -85,B 0,C 180,E1 -15507.582,E2 -15507.582} C_VEL
LIN {X 0,Y 336.718,Z 582.106,A -85,B 0,C 180,E1 -15507.778,E2 -15507.778} C_VEL
LIN {X 0,Y 334.924,Z 569.209,A -85,B 0,C 180,E1 -15508.889,E2 -15508.889} C_VEL
LIN {X 0,Y 332.21,Z 554.761,A -85,B 0,C 180,E1 -15510.404,E2 -15510.404} C_VEL
LIN {X 0,Y 331.836,Z 552.612,A -85,B 0,C 180,E1 -15510.663,E2 -15510.663} C_VEL
LIN {X 0,Y 332.515,Z 549.269,A -85,B 0,C 180,E1 -15511.382,E2 -15511.382} C_VEL
LIN {X 0,Y 332.08,Z 543.869,A -85,B 0,C 180,E1 -15513.006,E2 -15513.006} C_VEL
LIN {X 0,Y 331.096,Z 537.518,A -85,B 0,C 180,E1 -15515.288,E2 -15515.288} C_VEL
LIN {X 0,Y 330.225,Z 533.449,A -85,B 0,C 180,E1 -15517.044,E2 -15517.044} C_VEL
LIN {X 0,Y 329.002,Z 528.508,A -85,B 0,C 180,E1 -15519.734,E2 -15519.734} C_VEL
LIN {X 0,Y 328.302,Z 526.122,A -85,B 0,C 180,E1 -15521.577,E2 -15521.577} C_VEL
LIN {X 0,Y 327.884,Z 524.474,A -85,B 0,C 180,E1 -15523.307,E2 -15523.307} C_VEL
LIN {X 0,Y 327.636,Z 523.528,A -85,B 0,C 180,E1 -15525.062,E2 -15525.062} C_VEL
LIN {X 0,Y 327.761,Z 523.142,A -85,B 0,C 180,E1 -15526.806,E2 -15526.806} C_VEL
LIN {X 0,Y 328.204,Z 523.439,A -85,B 0,C 180,E1 -15528.545,E2 -15528.545} C_VEL
LIN {X 0,Y 328.976,Z 524.42,A -85,B 0,C 180,E1 -15530.271,E2 -15530.271} C_VEL
LIN {X 0,Y 331.141,Z 527.128,A -85,B 0,C 180,E1 -15532.952,E2 -15532.952} C_VEL
LIN {X 0,Y 332.795,Z 530.16,A -85,B 0,C 180,E1 -15534.641,E2 -15534.641} C_VEL
LIN {X 0,Y 333.537,Z 531.782,A -85,B 0,C 180,E1 -15535.325,E2 -15535.325} C_VEL
LIN {X 0,Y 334.761,Z 540.78,A -85,B 0,C 180,E1 -15537.525,E2 -15537.525} C_VEL
LIN {X 0,Y 335.753,Z 546.616,A -85,B 0,C 180,E1 -15538.741,E2 -15538.741} C_VEL
LIN {X 0,Y 335.684,Z 550.043,A -85,B 0,C 180,E1 -15539.231,E2 -15539.231} C_VEL
LIN {X 0,Y 334.702,Z 559.128,A -85,B 0,C 180,E1 -15540.165,E2 -15540.165} C_VEL
LIN {X 0,Y 334.91,Z 565.038,A -85,B 0,C 180,E1 -15540.575,E2 -15540.575} C_VEL
LIN {X 0,Y 326.505,Z 656.219,A -85,B 0,C 180,E1 -15544.201,E2 -15544.201} C_VEL
LIN {X 0,Y 324.693,Z 680.302,A -85,B 0,C 180,E1 -15545.205,E2 -15545.205} C_VEL
LIN {X 0,Y 323.53,Z 692.826,A -85,B 0,C 180,E1 -15545.957,E2 -15545.957} C_VEL
LIN {X 0,Y 322.162,Z 704.533,A -85,B 0,C 180,E1 -15546.879,E2 -15546.879} C_VEL
LIN {X 0,Y 320.558,Z 717.02,A -85,B 0,C 180,E1 -15548.117,E2 -15548.117} C_VEL
LIN {X 0,Y 318.714,Z 728.297,A -85,B 0,C 180,E1 -15549.509,E2 -15549.509} C_VEL
LIN {X 0,Y 316.83,Z 739.588,A -85,B 0,C 180,E1 -15551.238,E2 -15551.238} C_VEL
LIN {X 0,Y 315.121,Z 749.472,A -85,B 0,C 180,E1 -15553.146,E2 -15553.146} C_VEL
LIN {X 0,Y 313.785,Z 757.563,A -85,B 0,C 180,E1 -15555.074,E2 -15555.074} C_VEL
LIN {X 0,Y 312.674,Z 764.114,A -85,B 0,C 180,E1 -15557.011,E2 -15557.011} C_VEL
LIN {X 0,Y 311.855,Z 769.352,A -85,B 0,C 180,E1 -15558.956,E2 -15558.956} C_VEL
LIN {X 0,Y 311.283,Z 773.449,A -85,B 0,C 180,E1 -15560.907,E2 -15560.907} C_VEL
LIN {X 0,Y 310.998,Z 775.581,A -85,B 0,C 180,E1 -15562.207,E2 -15562.207} C_VEL
LIN {X 0,Y 310.801,Z 777.99,A -85,B 0,C 180,E1 -15564.241,E2 -15564.241} C_VEL
LIN {X 0,Y 310.702,Z 779.247,A -85,B 0,C 180,E1 -15566.109,E2 -15566.109} C_VEL
LIN {X 0,Y 310.706,Z 779.606,A -85,B 0,C 180,E1 -15567.407,E2 -15567.407} C_VEL
LIN {X 0,Y 310.708,Z 779.486,A -85,B 0,C 180,E1 -15568.704,E2 -15568.704} C_VEL
LIN {X 0,Y 310.675,Z 780.517,A -85,B 0,C 180,E1 -15571.296,E2 -15571.296} C_VEL
LIN {X 0,Y 310.684,Z 780.566,A -85,B 0,C 180,E1 -15572.593,E2 -15572.593} C_VEL
LIN {X 0,Y 310.696,Z 779.55,A -85,B 0,C 180,E1 -15575.191,E2 -15575.191} C_VEL
LIN {X 0,Y 310.996,Z 777.076,A -85,B 0,C 180,E1 -15577.793,E2 -15577.793} C_VEL
LIN {X 0,Y 311.597,Z 773.109,A -85,B 0,C 180,E1 -15580.395,E2 -15580.395} C_VEL
LIN {X 0,Y 312.335,Z 769.064,A -85,B 0,C 180,E1 -15582.343,E2 -15582.343} C_VEL
LIN {X 0,Y 313.471,Z 764.077,A -85,B 0,C 180,E1 -15584.278,E2 -15584.278} C_VEL
LIN {X 0,Y 314.978,Z 756.887,A -85,B 0,C 180,E1 -15586.53,E2 -15586.53} C_VEL
LIN {X 0,Y 317.005,Z 748.035,A -85,B 0,C 180,E1 -15588.752,E2 -15588.752} C_VEL
LIN {X 0,Y 319.178,Z 738.85,A -85,B 0,C 180,E1 -15590.629,E2 -15590.629} C_VEL
LIN {X 0,Y 321.685,Z 727.783,A -85,B 0,C 180,E1 -15592.478,E2 -15592.478} C_VEL
LIN {X 0,Y 324.138,Z 716.625,A -85,B 0,C 180,E1 -15593.988,E2 -15593.988} C_VEL
LIN {X 0,Y 326.723,Z 703.921,A -85,B 0,C 180,E1 -15595.385,E2 -15595.385} C_VEL
LIN {X 0,Y 328.888,Z 691.496,A -85,B 0,C 180,E1 -15596.492,E2 -15596.492} C_VEL
LIN {X 0,Y 331.07,Z 678.024,A -85,B 0,C 180,E1 -15597.412,E2 -15597.412} C_VEL
LIN {X 0,Y 332.902,Z 662.947,A -85,B 0,C 180,E1 -15598.188,E2 -15598.188} C_VEL
LIN {X 0,Y 341.073,Z 576.231,A -85,B 0,C 180,E1 -15601.231,E2 -15601.231} C_VEL
LIN {X 0,Y 342.178,Z 565.187,A -85,B 0,C 180,E1 -15601.637,E2 -15601.637} C_VEL
LIN {X 0,Y 341.389,Z 558.011,A -85,B 0,C 180,E1 -15602.23,E2 -15602.23} C_VEL
LIN {X 0,Y 337.818,Z 550.85,A -85,B 0,C 180,E1 -15603.543,E2 -15603.543} C_VEL
LIN {X 0,Y 335.528,Z 546.74,A -85,B 0,C 180,E1 -15604.44,E2 -15604.44} C_VEL
LIN {X 0,Y 333.276,Z 542.858,A -85,B 0,C 180,E1 -15605.392,E2 -15605.392} C_VEL
LIN {X 0,Y 330.025,Z 537.923,A -85,B 0,C 180,E1 -15606.915,E2 -15606.915} C_VEL
LIN {X 0,Y 326.415,Z 532.75,A -85,B 0,C 180,E1 -15609.062,E2 -15609.062} C_VEL
LIN {X 0,Y 325.721,Z 530.258,A -85,B 0,C 180,E1 -15611.981,E2 -15611.981} C_VEL
LIN {X 0,Y 325.353,Z 529.275,A -85,B 0,C 180,E1 -15614.534,E2 -15614.534} C_VEL
LIN {X 0,Y 325.367,Z 529.341,A -85,B 0,C 180,E1 -15617.258,E2 -15617.258} C_VEL
LIN {X 0,Y 325.613,Z 530.366,A -85,B 0,C 180,E1 -15619.645,E2 -15619.645} C_VEL
LIN {X 0,Y 326.253,Z 533.237,A -85,B 0,C 180,E1 -15622.849,E2 -15622.849} C_VEL
LIN {X 0,Y 327.074,Z 536.42,A -85,B 0,C 180,E1 -15625.177,E2 -15625.177} C_VEL
LIN {X 0,Y 331.048,Z 543.461,A -85,B 0,C 180,E1 -15627.418,E2 -15627.418} C_VEL
LIN {X 0,Y 334.252,Z 549.628,A -85,B 0,C 180,E1 -15628.938,E2 -15628.938} C_VEL
LIN {X 0,Y 336.333,Z 554.212,A -85,B 0,C 180,E1 -15629.872,E2 -15629.872} C_VEL
LIN {X 0,Y 337.68,Z 561.305,A -85,B 0,C 180,E1 -15630.714,E2 -15630.714} C_VEL
LIN {X 0,Y 339.353,Z 572.925,A -85,B 0,C 180,E1 -15631.883,E2 -15631.883} C_VEL
LIN {X 0,Y 340.151,Z 582.696,A -85,B 0,C 180,E1 -15632.672,E2 -15632.672} C_VEL
LIN {X 0,Y 331.924,Z 659.189,A -85,B 0,C 180,E1 -15635.697,E2 -15635.697} C_VEL
LIN {X 0,Y 330.276,Z 672.178,A -85,B 0,C 180,E1 -15636.43,E2 -15636.43} C_VEL
LIN {X 0,Y 328.116,Z 685.841,A -85,B 0,C 180,E1 -15637.453,E2 -15637.453} C_VEL
LIN {X 0,Y 325.915,Z 698.304,A -85,B 0,C 180,E1 -15638.661,E2 -15638.661} C_VEL
LIN {X 0,Y 323.414,Z 710.634,A -85,B 0,C 180,E1 -15640.151,E2 -15640.151} C_VEL
LIN {X 0,Y 320.963,Z 721.704,A -85,B 0,C 180,E1 -15641.819,E2 -15641.819} C_VEL
LIN {X 0,Y 318.612,Z 731.454,A -85,B 0,C 180,E1 -15643.666,E2 -15643.666} C_VEL
LIN {X 0,Y 316.76,Z 739.486,A -85,B 0,C 180,E1 -15645.546,E2 -15645.546} C_VEL
LIN {X 0,Y 315.384,Z 744.994,A -85,B 0,C 180,E1 -15647.124,E2 -15647.124} C_VEL
LIN {X 0,Y 313.961,Z 750.423,A -85,B 0,C 180,E1 -15649.031,E2 -15649.031} C_VEL
LIN {X 0,Y 312.938,Z 754.714,A -85,B 0,C 180,E1 -15650.955,E2 -15650.955} C_VEL
LIN {X 0,Y 312.35,Z 756.993,A -85,B 0,C 180,E1 -15652.241,E2 -15652.241} C_VEL
LIN {X 0,Y 311.774,Z 758.799,A -85,B 0,C 180,E1 -15653.528,E2 -15653.528} C_VEL
LIN {X 0,Y 311.417,Z 760.134,A -85,B 0,C 180,E1 -15654.821,E2 -15654.821} C_VEL
LIN {X 0,Y 311.206,Z 761.055,A -85,B 0,C 180,E1 -15656.115,E2 -15656.115} C_VEL
LIN {X 0,Y 310.993,Z 761.58,A -85,B 0,C 180,E1 -15657.409,E2 -15657.409} C_VEL
LIN {X 0,Y 310.819,Z 761.659,A -85,B 0,C 180,E1 -15658.704,E2 -15658.704} C_VEL
LIN {X 0,Y 310.728,Z 761.284,A -85,B 0,C 180,E1 -15660,E2 -15660} C_VEL
LIN {X 0,Y 310.699,Z 760.492,A -85,B 0,C 180,E1 -15661.296,E2 -15661.296} C_VEL
LIN {X 0,Y 310.735,Z 759.28,A -85,B 0,C 180,E1 -15662.593,E2 -15662.593} C_VEL
LIN {X 0,Y 310.76,Z 756.589,A -85,B 0,C 180,E1 -15664.54,E2 -15664.54} C_VEL
LIN {X 0,Y 310.939,Z 752.829,A -85,B 0,C 180,E1 -15666.489,E2 -15666.489} C_VEL
LIN {X 0,Y 311.2,Z 747.876,A -85,B 0,C 180,E1 -15668.441,E2 -15668.441} C_VEL
LIN {X 0,Y 311.628,Z 741.597,A -85,B 0,C 180,E1 -15670.394,E2 -15670.394} C_VEL
LIN {X 0,Y 312.252,Z 733.76,A -85,B 0,C 180,E1 -15672.346,E2 -15672.346} C_VEL
LIN {X 0,Y 313.115,Z 724.095,A -85,B 0,C 180,E1 -15674.294,E2 -15674.294} C_VEL
LIN {X 0,Y 313.81,Z 715.249,A -85,B 0,C 180,E1 -15675.756,E2 -15675.756} C_VEL
LIN {X 0,Y 314.891,Z 703.275,A -85,B 0,C 180,E1 -15677.368,E2 -15677.368} C_VEL
LIN {X 0,Y 315.943,Z 691.464,A -85,B 0,C 180,E1 -15678.649,E2 -15678.649} C_VEL
LIN {X 0,Y 316.847,Z 678.248,A -85,B 0,C 180,E1 -15679.771,E2 -15679.771} C_VEL
LIN {X 0,Y 317.721,Z 664.721,A -85,B 0,C 180,E1 -15680.643,E2 -15680.643} C_VEL
LIN {X 0,Y 318.455,Z 650.657,A -85,B 0,C 180,E1 -15681.27,E2 -15681.27} C_VEL
LIN {X 0,Y 321.285,Z 574.103,A -85,B 0,C 180,E1 -15683.781,E2 -15683.781} C_VEL
LIN {X 0,Y 317.106,Z 540.492,A -85,B 0,C 180,E1 -15685.16,E2 -15685.16} C_VEL
LIN {X 0,Y 317.008,Z 539.068,A -85,B 0,C 180,E1 -15685.227,E2 -15685.227} C_VEL
LIN {X 0,Y 318.665,Z 525.609,A -85,B 0,C 180,E1 -15688.382,E2 -15688.382} C_VEL
LIN {X 0,Y 317.294,Z 518.366,A -85,B 0,C 180,E1 -15690.248,E2 -15690.248} C_VEL
LIN {X 0,Y 314.17,Z 503.885,A -85,B 0,C 180,E1 -15694.137,E2 -15694.137} C_VEL
LIN {X 0,Y 312.565,Z 496.674,A -85,B 0,C 180,E1 -15696.18,E2 -15696.18} C_VEL
LIN {X 0,Y 312.506,Z 496.681,A -85,B 0,C 180,E1 -15700.125,E2 -15700.125} C_VEL
LIN {X 0,Y 312.514,Z 496.679,A -85,B 0,C 180,E1 -15702.427,E2 -15702.427} C_VEL
LIN {X 0,Y 312.46,Z 496.687,A -85,B 0,C 180,E1 -15706.035,E2 -15706.035} C_VEL
LIN {X 0,Y 312.505,Z 496.683,A -85,B 0,C 180,E1 -15709.874,E2 -15709.874} C_VEL
LIN {X 0,Y 312.537,Z 496.677,A -85,B 0,C 180,E1 -15714.05,E2 -15714.05} C_VEL
LIN {X 0,Y 312.506,Z 496.683,A -85,B 0,C 180,E1 -15717.334,E2 -15717.334} C_VEL
LIN {X 0,Y 312.553,Z 496.677,A -85,B 0,C 180,E1 -15721.276,E2 -15721.276} C_VEL
LIN {X 0,Y 312.587,Z 496.669,A -85,B 0,C 180,E1 -15724.711,E2 -15724.711} C_VEL
LIN {X 0,Y 312.589,Z 496.675,A -85,B 0,C 180,E1 -15727.529,E2 -15727.529} C_VEL
LIN {X 0,Y 312.64,Z 496.667,A -85,B 0,C 180,E1 -15731.656,E2 -15731.656} C_VEL
